KUKA KRL program: MyProgram_305().src

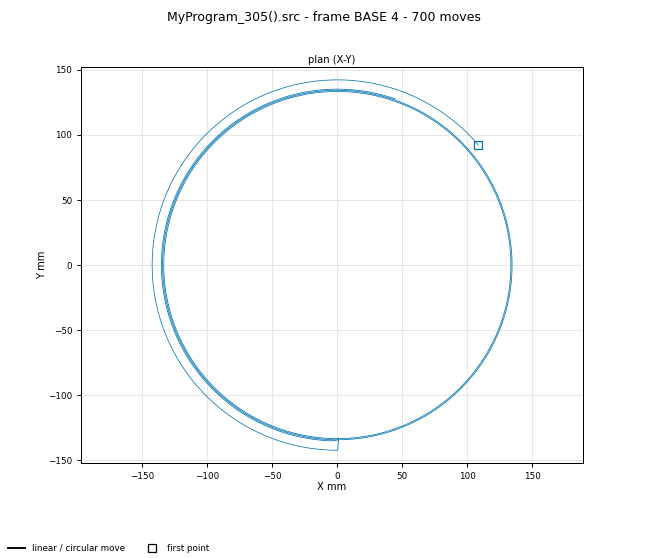
[picture p0: tool path of MyProgram_305().src in frame BASE 4, 700 of 700 moves have a stored position in this frame; points joined in program order, loops and branches not executed]
&ACCESS RVP
&REL 1
&PARAM TEMPLATE = C:\KRC\Roboter\Template\vorgabe
&PARAM EDITMASK = *
DEF MyProgram_305()
; ---- Setting reference (Base) ----
$BASE = BASE_DATA[4]

; --------------------------
; ---- Setting tool (TCP) ----
$TOOL = TOOL_DATA[3]
; --------------------------

$VEL.CP = VEL_APROX_PRINT
Startdeposition()
$VEL.CP = VEL_PRINT
LIN {X 108.497,Y 92.2361,Z 180,A 42.4872,B 5.0785,C 0.1519,E1 5.2028,E2 410.3593} C_DIS
LIN {X 105.629,Y 95.5075,Z 180,A 44.1909,B 5.0786,C 0.1489,E1 5.1996,E2 408.6614} C_DIS
LIN {X 103.133,Y 98.1976,Z 180,A 45.6374,B 5.0786,C 0.1462,E1 5.1969,E2 407.2184} C_DIS
LIN {X 100.1614,Y 101.227,Z 180,A 47.3328,B 5.0788,C 0.1429,E1 5.1935,E2 405.5242} C_DIS
LIN {X 97.4009,Y 103.8864,Z 180,A 48.922,B 5.0788,C 0.1392,E1 5.1903,E2 403.9286} C_DIS
LIN {X 93.8802,Y 107.0781,Z 180,A 50.7517,B 5.079,C 0.1367,E1 5.1865,E2 402.1093} C_DIS
LIN {X 90.8749,Y 109.6397,Z 180,A 52.3365,B 5.079,C 0.1338,E1 5.1831,E2 400.5248} C_DIS
LIN {X 87.4731,Y 112.3728,Z 180,A 54.072,B 5.0791,C 0.1309,E1 5.1793,E2 398.7918} C_DIS
LIN {X 84.1137,Y 114.9089,Z 180,A 55.7406,B 5.0791,C 0.1284,E1 5.1756,E2 397.1263} C_DIS
LIN {X 80.5548,Y 117.431,Z 180,A 57.3714,B 5.0791,C 0.1271,E1 5.1719,E2 395.5116} C_DIS
LIN {X 76.9953,Y 119.7953,Z 180,A 59.0501,B 5.0793,C 0.1249,E1 5.1679,E2 393.8381} C_DIS
LIN {X 73.811,Y 121.7829,Z 180,A 60.6088,B 5.0793,C 0.122,E1 5.1642,E2 392.273} C_DIS
LIN {X 70.1888,Y 123.9065,Z 180,A 62.306,B 5.0793,C 0.1195,E1 5.1601,E2 390.5749} C_DIS
LIN {X 66.4714,Y 125.9372,Z 180,A 63.6729,B 5.0793,C 0.1215,E1 5.1569,E2 389.2516} C_DIS
LIN {X 63.8622,Y 127.2826,Z 180,A 65.0425,B 5.0794,C 0.1175,E1 5.1534,E2 387.8578} C_DIS
LIN {X 60.0878,Y 129.1051,Z 180,A 66.7376,B 5.0794,C 0.1152,E1 5.1491,E2 386.1617} C_DIS
LIN {X 56.1086,Y 130.8838,Z 180,A 68.5245,B 5.0795,C 0.1128,E1 5.1445,E2 384.3707} C_DIS
LIN {X 51.5758,Y 132.7347,Z 180,A 70.4336,B 5.0795,C 0.1114,E1 5.1396,E2 382.4697} C_DIS
LIN {X 47.7101,Y 134.1742,Z 180,A 72.0661,B 5.0795,C 0.11,E1 5.1353,E2 380.841} C_DIS
LIN {X 44.2479,Y 135.3562,Z 180,A 73.5098,B 5.0796,C 0.109,E1 5.1315,E2 379.4014} C_DIS
LIN {X 40.4549,Y 136.5365,Z 180,A 75.105,B 5.0796,C 0.1077,E1 5.1272,E2 377.8068} C_DIS
LIN {X 36.267,Y 137.708,Z 180,A 76.8248,B 5.0796,C 0.1066,E1 5.1226,E2 376.0913} C_DIS
LIN {X 32.5455,Y 138.6366,Z 180,A 78.3403,B 5.0796,C 0.1059,E1 5.1185,E2 374.5798} C_DIS
LIN {X 29.1374,Y 139.3923,Z 180,A 79.7398,B 5.0797,C 0.105,E1 5.1147,E2 373.1814} C_DIS
LIN {X 26.0616,Y 139.9996,Z 180,A 80.976,B 5.0797,C 0.1046,E1 5.1113,E2 371.9487} C_DIS
LIN {X 22.184,Y 140.6651,Z 180,A 82.5487,B 5.0797,C 0.1039,E1 5.107,E2 370.3778} C_DIS
LIN {X 18.7998,Y 141.157,Z 180,A 83.9352,B 5.0797,C 0.1032,E1 5.1031,E2 368.9904} C_DIS
LIN {X 15.3344,Y 141.5752,Z 180,A 85.3305,B 5.0797,C 0.1028,E1 5.0993,E2 367.5967} C_DIS
LIN {X 11.8606,Y 141.9085,Z 180,A 86.7247,B 5.0797,C 0.1025,E1 5.0954,E2 366.2043} C_DIS
LIN {X 8.3796,Y 142.157,Z 180,A 88.0849,B 5.0797,C 0.1027,E1 5.0916,E2 364.8504} C_DIS
LIN {X 5.2259,Y 142.3077,Z 180,A 89.42,B 5.0797,C 0.1017,E1 5.0879,E2 363.5075} C_DIS
LIN {X 0.9091,Y 142.4005,Z 180,A 91.0268,B 5.0797,C 0.103,E1 5.0834,E2 361.9182} C_DIS
LIN {X -1.7521,Y 142.3939,Z 180,A 92.2232,B 5.0797,C 0.1016,E1 5.08,E2 360.7062} C_DIS
LIN {X -5.5962,Y 142.2933,Z 180,A 93.6931,B 5.0797,C 0.1025,E1 5.076,E2 359.2469} C_DIS
LIN {X -8.754,Y 142.1339,Z 180,A 95.0256,B 5.0797,C 0.102,E1 5.0722,E2 357.9071} C_DIS
LIN {X -12.2328,Y 141.877,Z 180,A 96.4261,B 5.0797,C 0.1023,E1 5.0683,E2 356.5077} C_DIS
LIN {X -15.7034,Y 141.5355,Z 180,A 97.8292,B 5.0797,C 0.1026,E1 5.0644,E2 355.1055} C_DIS
LIN {X -19.165,Y 141.1092,Z 180,A 99.3368,B 5.0797,C 0.1019,E1 5.0602,E2 353.5852} C_DIS
LIN {X -23.0175,Y 140.5312,Z 180,A 100.8267,B 5.0797,C 0.1034,E1 5.0561,E2 352.1061} C_DIS
LIN {X -26.1042,Y 139.9915,Z 180,A 102.0941,B 5.0797,C 0.1039,E1 5.0527,E2 350.8385} C_DIS
LIN {X -29.5153,Y 139.3118,Z 180,A 103.4975,B 5.0797,C 0.1046,E1 5.0488,E2 349.4354} C_DIS
LIN {X -33.0361,Y 138.5184,Z 180,A 104.9194,B 5.0797,C 0.1058,E1 5.045,E2 348.0183} C_DIS
LIN {X -36.6145,Y 137.6154,Z 180,A 106.458,B 5.0797,C 0.1062,E1 5.0408,E2 346.4736} C_DIS
LIN {X -40.0082,Y 136.6672,Z 180,A 107.8792,B 5.0797,C 0.1072,E1 5.037,E2 345.0529} C_DIS
LIN {X -43.347,Y 135.6452,Z 180,A 109.2169,B 5.0797,C 0.109,E1 5.0334,E2 343.7247} C_DIS
LIN {X -46.3341,Y 134.6545,Z 180,A 110.6489,B 5.0797,C 0.1084,E1 5.0296,E2 342.2722} C_DIS
LIN {X -49.9691,Y 133.3479,Z 180,A 112.1416,B 5.0796,C 0.1105,E1 5.0257,E2 340.7885} C_DIS
LIN {X -52.8929,Y 132.2159,Z 180,A 113.4133,B 5.0796,C 0.1117,E1 5.0224,E2 339.5163} C_DIS
LIN {X -56.1132,Y 130.8818,Z 180,A 114.9688,B 5.0796,C 0.1116,E1 5.0183,E2 337.942} C_DIS
LIN {X -60.2519,Y 129.0292,Z 180,A 116.7977,B 5.0796,C 0.1136,E1 5.0137,E2 336.1139} C_DIS
LIN {X -64.2345,Y 127.093,Z 180,A 118.4648,B 5.0794,C 0.117,E1 5.0096,E2 334.4628} C_DIS
LIN {X -67.29,Y 125.5037,Z 180,A 119.9727,B 5.0794,C 0.1176,E1 5.0058,E2 332.9403} C_DIS
LIN {X -70.8659,Y 123.5203,Z 180,A 121.6,B 5.0794,C 0.12,E1 5.0019,E2 331.3165} C_DIS
LIN {X -74.4835,Y 121.3727,Z 180,A 123.3149,B 5.0794,C 0.1222,E1 4.9978,E2 329.6} C_DIS
LIN {X -77.8009,Y 119.2738,Z 180,A 124.9752,B 5.0793,C 0.1238,E1 4.9938,E2 327.9305} C_DIS
LIN {X -81.4658,Y 116.8009,Z 180,A 126.8101,B 5.0793,C 0.1261,E1 4.9896,E2 326.0897} C_DIS
LIN {X -85.414,Y 113.9463,Z 180,A 128.7148,B 5.0791,C 0.1298,E1 4.9853,E2 324.1938} C_DIS
LIN {X -88.4535,Y 111.6027,Z 180,A 130.3727,B 5.0791,C 0.1314,E1 4.9817,E2 322.5224} C_DIS
LIN {X -92.2127,Y 108.5169,Z 180,A 132.2804,B 5.079,C 0.1354,E1 4.9776,E2 320.6226} C_DIS
LIN {X -95.5234,Y 105.6146,Z 180,A 134.0811,B 5.079,C 0.1385,E1 4.9738,E2 318.8196} C_DIS
LIN {X -98.7082,Y 102.645,Z 180,A 135.9095,B 5.0788,C 0.1411,E1 4.9701,E2 316.9829} C_DIS
LIN {X -101.7995,Y 99.5791,Z 180,A 137.6842,B 5.0788,C 0.1444,E1 4.9666,E2 315.2066} C_DIS
LIN {X -104.4911,Y 96.7516,Z 180,A 139.363,B 5.0787,C 0.1467,E1 4.9634,E2 313.515} C_DIS
LIN {X -107.2862,Y 93.6417,Z 180,A 140.9733,B 5.0785,C 0.1509,E1 4.9604,E2 311.9156} C_DIS
LIN {X -110.089,Y 90.3304,Z 180,A 142.8502,B 5.0785,C 0.1535,E1 4.957,E2 310.0231} C_DIS
LIN {X -112.7881,Y 86.9374,Z 180,A 144.5372,B 5.0783,C 0.1579,E1 4.9541,E2 308.345} C_DIS
LIN {X -115.4142,Y 83.4188,Z 180,A 146.4481,B 5.0783,C 0.1606,E1 4.9509,E2 306.4169} C_DIS
LIN {X -118.0164,Y 79.6949,Z 180,A 148.3219,B 5.0781,C 0.1645,E1 4.948,E2 304.5386} C_DIS
LIN {X -120.4113,Y 76.0279,Z 180,A 150.0764,B 5.078,C 0.1688,E1 4.9453,E2 302.7867} C_DIS
LIN {X -122.5944,Y 72.456,Z 180,A 151.8564,B 5.0779,C 0.172,E1 4.9428,E2 300.9958} C_DIS
LIN {X -124.8426,Y 68.5097,Z 180,A 153.5741,B 5.0777,C 0.1775,E1 4.9404,E2 299.2939} C_DIS
LIN {X -126.5036,Y 65.3923,Z 180,A 155.0584,B 5.0776,C 0.1805,E1 4.9385,E2 297.8026} C_DIS
LIN {X -128.0663,Y 62.2752,Z 180,A 156.662,B 5.0776,C 0.1824,E1 4.9365,E2 296.174} C_DIS
LIN {X -129.8361,Y 58.4918,Z 180,A 158.3236,B 5.0774,C 0.1869,E1 4.9346,E2 294.5162} C_DIS
LIN {X -131.6971,Y 54.1756,Z 180,A 160.1551,B 5.0772,C 0.1923,E1 4.9326,E2 292.6943} C_DIS
LIN {X -132.8628,Y 51.2461,Z 180,A 161.4663,B 5.077,C 0.1953,E1 4.9313,E2 291.3785} C_DIS
LIN {X -134.0776,Y 47.978,Z 180,A 162.9414,B 5.077,C 0.1985,E1 4.9298,E2 289.8952} C_DIS
LIN {X -135.2171,Y 44.6658,Z 180,A 164.3548,B 5.0768,C 0.2022,E1 4.9286,E2 288.4824} C_DIS
LIN {X -136.271,Y 41.3393,Z 180,A 165.7974,B 5.0766,C 0.2057,E1 4.9274,E2 287.0359} C_DIS
LIN {X -137.2431,Y 37.9877,Z 180,A 167.24,B 5.0765,C 0.2092,E1 4.9263,E2 285.5894} C_DIS
LIN {X -138.2216,Y 34.2642,Z 180,A 168.83,B 5.0763,C 0.2132,E1 4.9252,E2 283.9955} C_DIS
LIN {X -139.0703,Y 30.6335,Z 180,A 170.3234,B 5.0761,C 0.2174,E1 4.9243,E2 282.5042} C_DIS
LIN {X -139.7442,Y 27.3977,Z 180,A 171.7791,B 5.0761,C 0.22,E1 4.9235,E2 281.033} C_DIS
LIN {X -140.3142,Y 24.3143,Z 180,A 173.0378,B 5.0759,C 0.2236,E1 4.9228,E2 279.7758} C_DIS
LIN {X -140.9162,Y 20.5282,Z 180,A 174.6365,B 5.0757,C 0.2274,E1 4.9222,E2 278.1708} C_DIS
LIN {X -141.3751,Y 17.0814,Z 180,A 176.0816,B 5.0755,C 0.231,E1 4.9217,E2 276.7207} C_DIS
LIN {X -141.7543,Y 13.5793,Z 180,A 177.5278,B 5.0754,C 0.2348,E1 4.9212,E2 275.2719} C_DIS
LIN {X -142.0445,Y 10.1047,Z 180,A 178.9648,B 5.0752,C 0.2385,E1 4.9209,E2 273.8315} C_DIS
LIN {X -142.2324,Y 6.9769,Z 180,A -179.6803,B 5.0751,C 0.2412,E1 4.9207,E2 272.4651} C_DIS
LIN {X -142.3708,Y 3.1405,Z 180,A -178.0382,B 5.0749,C 0.2448,E1 4.9207,E2 270.8114} C_DIS
LIN {X -142.4071,Y -0.0245,Z 180,A -176.7476,B 5.0747,C 0.2483,E1 4.9207,E2 269.5195} C_DIS
LIN {X -142.3604,Y -3.5237,Z 180,A -175.2972,B 5.0746,C 0.2519,E1 4.9207,E2 268.0644} C_DIS
LIN {X -142.231,Y -7.0045,Z 180,A -173.9334,B 5.0743,C 0.2562,E1 4.9208,E2 266.7066} C_DIS
LIN {X -142.0173,Y -10.477,Z 180,A -172.4754,B 5.0742,C 0.2597,E1 4.9211,E2 265.2419} C_DIS
LIN {X -141.7082,Y -14.0595,Z 180,A -171.0171,B 5.074,C 0.2637,E1 4.9215,E2 263.7831} C_DIS
LIN {X -141.3237,Y -17.5129,Z 180,A -169.5808,B 5.0738,C 0.2673,E1 4.922,E2 262.3427} C_DIS
LIN {X -140.8041,Y -21.2862,Z 180,A -167.9868,B 5.0736,C 0.271,E1 4.9226,E2 260.7416} C_DIS
LIN {X -140.2364,Y -24.7488,Z 180,A -166.6703,B 5.0733,C 0.2758,E1 4.9232,E2 259.4386} C_DIS
LIN {X -139.6676,Y -27.7843,Z 180,A -165.2521,B 5.0733,C 0.2777,E1 4.924,E2 257.998} C_DIS
LIN {X -138.9437,Y -31.2015,Z 180,A -163.8091,B 5.073,C 0.2813,E1 4.9248,E2 256.5508} C_DIS
LIN {X -138.1369,Y -34.5977,Z 180,A -162.2841,B 5.0729,C 0.2841,E1 4.9259,E2 255.0107} C_DIS
LIN {X -137.1471,Y -38.3311,Z 180,A -160.7717,B 5.0726,C 0.2887,E1 4.927,E2 253.5046} C_DIS
LIN {X -136.1664,Y -41.681,Z 180,A -159.328,B 5.0724,C 0.2921,E1 4.9281,E2 252.0566} C_DIS
LIN {X -135.2162,Y -44.6685,Z 180,A -158.0324,B 5.0722,C 0.2952,E1 4.9293,E2 250.7571} C_DIS
LIN {X -133.9438,Y -48.3491,Z 180,A -156.423,B 5.072,C 0.299,E1 4.9308,E2 249.1429} C_DIS
LIN {X -132.7219,Y -51.6087,Z 180,A -155.0665,B 5.0718,C 0.3031,E1 4.9321,E2 247.793} C_DIS
LIN {X -131.5581,Y -54.5086,Z 180,A -153.6984,B 5.0716,C 0.3054,E1 4.9336,E2 246.4108} C_DIS
LIN {X -130.1902,Y -57.7,Z 180,A -152.2583,B 5.0714,C 0.3086,E1 4.9352,E2 244.9656} C_DIS
LIN {X -128.7297,Y -60.8892,Z 180,A -150.8166,B 5.0712,C 0.3119,E1 4.9369,E2 243.5205} C_DIS
LIN {X -127.1988,Y -64.0267,Z 180,A -149.3238,B 5.0711,C 0.3146,E1 4.9387,E2 242.0166} C_DIS
LIN {X -125.4914,Y -67.313,Z 180,A -147.7585,B 5.0709,C 0.3176,E1 4.9408,E2 240.4419} C_DIS
LIN {X -123.3746,Y -71.1188,Z 180,A -145.9254,B 5.0707,C 0.3211,E1 4.9433,E2 238.5986} C_DIS
LIN {X -121.1439,Y -74.8563,Z 180,A -144.1142,B 5.0704,C 0.3247,E1 4.946,E2 236.7801} C_DIS
LIN {X -118.8861,Y -78.3915,Z 180,A -142.4947,B 5.0701,C 0.3293,E1 4.9484,E2 235.1704} C_DIS
LIN {X -116.4277,Y -81.9983,Z 180,A -140.6547,B 5.0699,C 0.3325,E1 4.9514,E2 233.3197} C_DIS
LIN {X -113.8558,Y -85.534,Z 180,A -138.8009,B 5.0697,C 0.3356,E1 4.9545,E2 231.4538} C_DIS
LIN {X -111.0721,Y -89.1192,Z 180,A -136.9271,B 5.0695,C 0.3391,E1 4.9577,E2 229.5741} C_DIS
LIN {X -108.1727,Y -92.6172,Z 180,A -135.0822,B 5.0692,C 0.3428,E1 4.9611,E2 227.7274} C_DIS
LIN {X -105.043,Y -96.1518,Z 180,A -133.218,B 5.069,C 0.347,E1 4.9645,E2 225.8684} C_DIS
LIN {X -102.3499,Y -99.0132,Z 180,A -131.546,B 5.0688,C 0.3492,E1 4.9678,E2 224.1844} C_DIS
LIN {X -98.9579,Y -102.4034,Z 180,A -129.6209,B 5.0685,C 0.353,E1 4.9716,E2 222.2603} C_DIS
LIN {X -95.6326,Y -105.5155,Z 180,A -127.7753,B 5.0683,C 0.3562,E1 4.9754,E2 220.4133} C_DIS
LIN {X -92.4851,Y -108.2854,Z 180,A -126.016,B 5.0682,C 0.3585,E1 4.9791,E2 218.6444} C_DIS
LIN {X -88.9817,Y -111.1824,Z 180,A -124.179,B 5.0679,C 0.3616,E1 4.9831,E2 216.8065} C_DIS
LIN {X -85.5169,Y -113.8687,Z 180,A -122.4297,B 5.0677,C 0.3646,E1 4.987,E2 215.0594} C_DIS
LIN {X -82.7018,Y -115.929,Z 180,A -120.8841,B 5.0677,C 0.3653,E1 4.9906,E2 213.4946} C_DIS
LIN {X -78.9676,Y -118.5042,Z 180,A -119.1549,B 5.0674,C 0.3691,E1 4.9945,E2 211.7785} C_DIS
LIN {X -75.4545,Y -120.7717,Z 180,A -117.4099,B 5.0673,C 0.3708,E1 4.9987,E2 210.025} C_DIS
LIN {X -71.7041,Y -123.0358,Z 180,A -115.6316,B 5.0671,C 0.373,E1 5.0029,E2 208.2445} C_DIS
LIN {X -68.4223,Y -124.8903,Z 180,A -114.1736,B 5.0669,C 0.3756,E1 5.0065,E2 206.7944} C_DIS
LIN {X -65.4161,Y -126.4913,Z 180,A -112.7306,B 5.0669,C 0.3765,E1 5.0101,E2 205.3415} C_DIS
LIN {X -62.2971,Y -128.0555,Z 180,A -111.1595,B 5.0669,C 0.3763,E1 5.0141,E2 203.7473} C_DIS
LIN {X -58.3478,Y -129.9004,Z 180,A -109.479,B 5.0667,C 0.379,E1 5.0183,E2 202.0767} C_DIS
LIN {X -54.1627,Y -131.7025,Z 180,A -107.7004,B 5.0665,C 0.3814,E1 5.0229,E2 200.3054} C_DIS
LIN {X -51.0763,Y -132.9289,Z 180,A -106.3426,B 5.0665,C 0.3824,E1 5.0264,E2 198.9443} C_DIS
LIN {X -47.7687,Y -134.1531,Z 180,A -104.8979,B 5.0663,C 0.3833,E1 5.0302,E2 197.4959} C_DIS
LIN {X -44.4743,Y -135.2809,Z 180,A -103.5072,B 5.0663,C 0.3845,E1 5.0339,E2 196.1064} C_DIS
LIN {X -41.0445,Y -136.3612,Z 180,A -102.061,B 5.0662,C 0.3856,E1 5.0378,E2 194.6599} C_DIS
LIN {X -37.9589,Y -137.2512,Z 180,A -100.7471,B 5.0662,C 0.3861,E1 5.0413,E2 193.3426} C_DIS
LIN {X -34.247,Y -138.2259,Z 180,A -99.1966,B 5.0661,C 0.387,E1 5.0455,E2 191.7909} C_DIS
LIN {X -30.8491,Y -139.0238,Z 180,A -97.7718,B 5.0661,C 0.3874,E1 5.0494,E2 190.3629} C_DIS
LIN {X -27.4327,Y -139.7375,Z 180,A -96.4289,B 5.0659,C 0.3888,E1 5.053,E2 189.0279} C_DIS
LIN {X -24.3325,Y -140.3109,Z 180,A -95.1056,B 5.0659,C 0.3886,E1 5.0567,E2 187.6967} C_DIS
LIN {X -20.5341,Y -140.9154,Z 180,A -93.538,B 5.0659,C 0.3888,E1 5.061,E2 186.1258} C_DIS
LIN {X -17.0731,Y -141.3761,Z 180,A -92.1332,B 5.0659,C 0.3892,E1 5.0649,E2 184.7205} C_DIS
LIN {X -13.6034,Y -141.752,Z 180,A -90.7314,B 5.0659,C 0.3894,E1 5.0688,E2 183.3185} C_DIS
LIN {X -10.1088,Y -142.0442,Z 180,A -89.3263,B 5.0659,C 0.3896,E1 5.0727,E2 181.9136} C_DIS
LIN {X -6.975,Y -142.2325,Z 180,A -88.0242,B 5.0659,C 0.3892,E1 5.0764,E2 180.6056} C_DIS
LIN {X -3.1346,Y -142.3709,Z 180,A -86.5457,B 5.0659,C 0.3899,E1 5.0805,E2 179.1357} C_DIS
LIN {X 0.3576,Y -142.4035,Z 180,A -85.1921,B 5.0659,C 0.3904,E1 5.0843,E2 177.7885} C_DIS
LIN {X 0.3576,Y -142.4035,Z 180,A -85.1921,B 5.0659,C 0.3904,E1 5.0843,E2 177.7885} C_DIS
Enddeposition()
LIN {X 0.9666,Y -133.4651,Z 181,A -85.2276,B 5.1404,C 0.3663,E1 5.1577,E2 177.5189} C_DIS
Startdeposition()
$VEL.CP = VEL_PRINT
LIN {X -2.5839,Y -133.4454,Z 181,A -87.4468,B 5.1398,C 0.3744,E1 5.1512,E2 179.8265} C_DIS
LIN {X -7.4832,Y -133.2619,Z 181,A -89.3757,B 5.14,C 0.3724,E1 5.1459,E2 181.7343} C_DIS
LIN {X -10.7403,Y -133.0379,Z 181,A -90.8246,B 5.14,C 0.3728,E1 5.1419,E2 183.1897} C_DIS
LIN {X -13.9556,Y -132.7386,Z 181,A -92.3357,B 5.1399,C 0.374,E1 5.1376,E2 184.717} C_DIS
LIN {X -17.9739,Y -132.2555,Z 181,A -93.9306,B 5.14,C 0.372,E1 5.1332,E2 186.2947} C_DIS
LIN {X -21.21,Y -131.7759,Z 181,A -95.3324,B 5.14,C 0.3716,E1 5.1294,E2 187.6966} C_DIS
LIN {X -25.2351,Y -131.0625,Z 181,A -97.1246,B 5.14,C 0.3713,E1 5.1244,E2 189.4941} C_DIS
LIN {X -29.2391,Y -130.2285,Z 181,A -98.8863,B 5.1401,C 0.3705,E1 5.1196,E2 191.257} C_DIS
LIN {X -33.132,Y -129.2923,Z 181,A -100.6252,B 5.1401,C 0.3698,E1 5.1149,E2 192.999} C_DIS
LIN {X -36.6436,Y -128.3429,Z 181,A -102.1754,B 5.1403,C 0.3687,E1 5.1107,E2 194.5482} C_DIS
LIN {X -39.6132,Y -127.4568,Z 181,A -103.5231,B 5.1403,C 0.3679,E1 5.1071,E2 195.8983} C_DIS
LIN {X -42.7923,Y -126.4253,Z 181,A -104.963,B 5.1403,C 0.3668,E1 5.1033,E2 197.3391} C_DIS
LIN {X -45.8064,Y -125.3643,Z 181,A -106.3383,B 5.1405,C 0.3657,E1 5.0997,E2 198.7152} C_DIS
LIN {X -48.9062,Y -124.1879,Z 181,A -107.7863,B 5.1405,C 0.3647,E1 5.0959,E2 200.1665} C_DIS
LIN {X -51.9332,Y -122.9525,Z 181,A -109.3465,B 5.1405,C 0.3649,E1 5.0918,E2 201.7464} C_DIS
LIN {X -55.582,Y -121.3464,Z 181,A -110.979,B 5.1407,C 0.3623,E1 5.0877,E2 203.3693} C_DIS
LIN {X -59.1813,Y -119.6314,Z 181,A -112.6628,B 5.1409,C 0.3601,E1 5.0835,E2 205.0497} C_DIS
LIN {X -62.0962,Y -118.1445,Z 181,A -114.0309,B 5.141,C 0.358,E1 5.0801,E2 206.4134} C_DIS
LIN {X -65.1789,Y -116.4748,Z 181,A -115.6023,B 5.141,C 0.3568,E1 5.0762,E2 207.9933} C_DIS
LIN {X -68.6256,Y -114.4782,Z 181,A -117.3443,B 5.1412,C 0.3548,E1 5.072,E2 209.7393} C_DIS
LIN {X -71.4102,Y -112.7619,Z 181,A -118.7665,B 5.1413,C 0.353,E1 5.0686,E2 211.1637} C_DIS
LIN {X -74.1524,Y -110.9776,Z 181,A -120.1893,B 5.1415,C 0.3511,E1 5.0653,E2 212.5887} C_DIS
LIN {X -76.849,Y -109.1277,Z 181,A -121.6122,B 5.1416,C 0.3492,E1 5.062,E2 214.014} C_DIS
LIN {X -80.0734,Y -106.785,Z 181,A -123.463,B 5.1417,C 0.3477,E1 5.0578,E2 215.8821} C_DIS
LIN {X -83.4049,Y -104.2035,Z 181,A -125.2703,B 5.1419,C 0.3447,E1 5.0539,E2 217.6889} C_DIS
LIN {X -86.7642,Y -101.4237,Z 181,A -127.2201,B 5.1421,C 0.3421,E1 5.0497,E2 219.6481} C_DIS
LIN {X -89.9135,Y -98.6421,Z 181,A -129.0282,B 5.1423,C 0.3389,E1 5.0459,E2 221.4565} C_DIS
LIN {X -92.8898,Y -95.8442,Z 181,A -130.7944,B 5.1425,C 0.3357,E1 5.0423,E2 223.2239} C_DIS
LIN {X -96.0008,Y -92.728,Z 181,A -132.7649,B 5.1427,C 0.3327,E1 5.0385,E2 225.204} C_DIS
LIN {X -98.8906,Y -89.6397,Z 181,A -134.5787,B 5.1429,C 0.329,E1 5.035,E2 227.0171} C_DIS
LIN {X -101.5992,Y -86.5577,Z 181,A -136.389,B 5.1431,C 0.3258,E1 5.0317,E2 228.833} C_DIS
LIN {X -104.1703,Y -83.4465,Z 181,A -138.1887,B 5.1433,C 0.3227,E1 5.0285,E2 230.6405} C_DIS
LIN {X -106.7734,Y -80.0887,Z 181,A -139.9426,B 5.1436,C 0.3181,E1 5.0256,E2 232.3851} C_DIS
LIN {X -109.129,Y -76.8471,Z 181,A -141.5517,B 5.1439,C 0.3132,E1 5.023,E2 233.9799} C_DIS
LIN {X -110.581,Y -74.7426,Z 181,A -142.819,B 5.1439,C 0.3122,E1 5.0209,E2 235.2678} C_DIS
LIN {X -112.3784,Y -72.0119,Z 181,A -144.2543,B 5.1442,C 0.3091,E1 5.0187,E2 236.7065} C_DIS
LIN {X -114.1093,Y -69.2367,Z 181,A -145.7239,B 5.1443,C 0.3064,E1 5.0166,E2 238.1836} C_DIS
LIN {X -116.1638,Y -65.7323,Z 181,A -147.4769,B 5.1446,C 0.3022,E1 5.0141,E2 239.937} C_DIS
LIN {X -117.724,Y -62.8949,Z 181,A -148.9275,B 5.1447,C 0.2993,E1 5.0122,E2 241.3944} C_DIS
LIN {X -119.2188,Y -60.0109,Z 181,A -150.327,B 5.1449,C 0.2959,E1 5.0104,E2 242.794} C_DIS
LIN {X -120.6574,Y -57.0626,Z 181,A -151.7847,B 5.1451,C 0.2927,E1 5.0086,E2 244.257} C_DIS
LIN {X -122.0201,Y -54.0867,Z 181,A -153.225,B 5.1453,C 0.2894,E1 5.007,E2 245.7009} C_DIS
LIN {X -123.3091,Y -51.0793,Z 181,A -154.6658,B 5.1455,C 0.2861,E1 5.0054,E2 247.1454} C_DIS
LIN {X -124.5313,Y -48.0227,Z 181,A -156.1156,B 5.1457,C 0.2827,E1 5.0039,E2 248.5989} C_DIS
LIN {X -125.9117,Y -44.2797,Z 181,A -157.8719,B 5.1459,C 0.2785,E1 5.0023,E2 250.3596} C_DIS
LIN {X -126.9576,Y -41.1855,Z 181,A -159.3753,B 5.1461,C 0.2755,E1 5.0009,E2 251.8746} C_DIS
LIN {X -128.1864,Y -37.1818,Z 181,A -161.2845,B 5.1463,C 0.2715,E1 4.9994,E2 253.7963} C_DIS
LIN {X -129.2875,Y -33.151,Z 181,A -163.0071,B 5.1466,C 0.2661,E1 4.9982,E2 255.5091} C_DIS
LIN {X -130.1807,Y -29.4485,Z 181,A -164.7066,B 5.1468,C 0.2621,E1 4.9971,E2 257.2155} C_DIS
LIN {X -130.9066,Y -26.0376,Z 181,A -166.2181,B 5.147,C 0.2581,E1 4.9962,E2 258.7278} C_DIS
LIN {X -131.5065,Y -22.8186,Z 181,A -167.6603,B 5.1472,C 0.2544,E1 4.9955,E2 260.1737} C_DIS
LIN {X -132.1563,Y -18.6798,Z 181,A -169.4876,B 5.1474,C 0.2496,E1 4.9947,E2 262.0032} C_DIS
LIN {X -132.5766,Y -15.4201,Z 181,A -171.1167,B 5.1474,C 0.2473,E1 4.9942,E2 263.6578} C_DIS
LIN {X -133.0382,Y -10.7366,Z 181,A -173.0667,B 5.1478,C 0.2411,E1 4.9937,E2 265.5978} C_DIS
LIN {X -133.2626,Y -7.4715,Z 181,A -174.576,B 5.1479,C 0.2379,E1 4.9934,E2 267.1188} C_DIS
LIN {X -133.4086,Y -4.0606,Z 181,A -176.1459,B 5.1481,C 0.2345,E1 4.9933,E2 268.7002} C_DIS
LIN {X -133.471,Y -0.1546,Z 181,A -177.6609,B 5.1484,C 0.2285,E1 4.9933,E2 270.1944} C_DIS
LIN {X -133.4459,Y 2.559,Z 181,A -179.0776,B 5.1484,C 0.2272,E1 4.9933,E2 271.6406} C_DIS
LIN {X -133.2634,Y 7.4588,Z 181,A 178.9282,B 5.1487,C 0.2203,E1 4.9935,E2 273.6199} C_DIS
LIN {X -133.0792,Y 10.2167,Z 181,A 177.5657,B 5.1488,C 0.2183,E1 4.9938,E2 275.0026} C_DIS
LIN {X -132.6571,Y 14.7129,Z 181,A 175.6954,B 5.1491,C 0.2123,E1 4.9943,E2 276.8631} C_DIS
LIN {X -132.2572,Y 17.9613,Z 181,A 174.2524,B 5.1492,C 0.2086,E1 4.9949,E2 278.3096} C_DIS
LIN {X -131.7782,Y 21.1963,Z 181,A 172.8099,B 5.1494,C 0.205,E1 4.9955,E2 279.7557} C_DIS
LIN {X -131.0459,Y 25.3219,Z 181,A 170.9461,B 5.1495,C 0.2004,E1 4.9964,E2 281.6259} C_DIS
LIN {X -130.2225,Y 29.2653,Z 181,A 169.1614,B 5.1497,C 0.196,E1 4.9975,E2 283.4158} C_DIS
LIN {X -129.289,Y 33.1449,Z 181,A 167.3853,B 5.1499,C 0.1918,E1 4.9987,E2 285.198} C_DIS
LIN {X -128.1873,Y 37.1787,Z 181,A 165.4197,B 5.1499,C 0.1882,E1 5.0002,E2 287.1825} C_DIS
LIN {X -126.959,Y 41.1809,Z 181,A 163.7112,B 5.1502,C 0.1826,E1 5.0016,E2 288.8789} C_DIS
LIN {X -125.9133,Y 44.2753,Z 181,A 162.2771,B 5.1503,C 0.1791,E1 5.0029,E2 290.3157} C_DIS
LIN {X -124.8551,Y 47.1748,Z 181,A 160.8879,B 5.1504,C 0.1761,E1 5.0042,E2 291.7113} C_DIS
LIN {X -123.5866,Y 50.4058,Z 181,A 159.3862,B 5.1506,C 0.1722,E1 5.0058,E2 293.2132} C_DIS
LIN {X -122.3894,Y 53.2448,Z 181,A 157.9942,B 5.1506,C 0.1693,E1 5.0073,E2 294.6123} C_DIS
LIN {X -120.6575,Y 57.0624,Z 181,A 156.0942,B 5.1508,C 0.1654,E1 5.0096,E2 296.5227} C_DIS
LIN {X -118.8877,Y 60.6613,Z 181,A 154.4056,B 5.1509,C 0.1608,E1 5.0117,E2 298.2059} C_DIS
LIN {X -117.2734,Y 63.7307,Z 181,A 152.8842,B 5.151,C 0.1573,E1 5.0137,E2 299.73} C_DIS
LIN {X -115.6804,Y 66.5791,Z 181,A 151.3012,B 5.151,C 0.1553,E1 5.0159,E2 301.3335} C_DIS
LIN {X -113.6413,Y 70.0023,Z 181,A 149.6873,B 5.1512,C 0.1504,E1 5.0182,E2 302.9344} C_DIS
LIN {X -111.8949,Y 72.7609,Z 181,A 148.2543,B 5.1513,C 0.1473,E1 5.0204,E2 304.3699} C_DIS
LIN {X -110.0603,Y 75.5072,Z 181,A 146.8037,B 5.1514,C 0.1442,E1 5.0226,E2 305.8232} C_DIS
LIN {X -108.1693,Y 78.1923,Z 181,A 145.3636,B 5.1514,C 0.1412,E1 5.025,E2 307.2657} C_DIS
LIN {X -106.221,Y 80.8197,Z 181,A 143.8414,B 5.1516,C 0.139,E1 5.0276,E2 308.8006} C_DIS
LIN {X -103.6931,Y 84.0383,Z 181,A 142.0294,B 5.1516,C 0.1356,E1 5.0307,E2 310.6176} C_DIS
LIN {X -101.06,Y 87.1866,Z 181,A 140.268,B 5.1517,C 0.1318,E1 5.0339,E2 312.3775} C_DIS
LIN {X -98.341,Y 90.2422,Z 181,A 138.4627,B 5.1518,C 0.1285,E1 5.0373,E2 314.1872} C_DIS
LIN {X -95.5305,Y 93.2129,Z 181,A 136.6586,B 5.1519,C 0.1253,E1 5.0408,E2 315.9956} C_DIS
LIN {X -92.6287,Y 96.0969,Z 181,A 134.8509,B 5.1519,C 0.1223,E1 5.0444,E2 317.8079} C_DIS
LIN {X -89.6302,Y 98.8991,Z 181,A 133.0781,B 5.1521,C 0.119,E1 5.048,E2 319.5805} C_DIS
LIN {X -86.5579,Y 101.599,Z 181,A 131.2764,B 5.1521,C 0.1162,E1 5.0519,E2 321.3862} C_DIS
LIN {X -83.4037,Y 104.2044,Z 181,A 129.4735,B 5.1521,C 0.1135,E1 5.0558,E2 323.1932} C_DIS
LIN {X -80.2142,Y 106.6787,Z 181,A 127.7852,B 5.1522,C 0.1101,E1 5.0595,E2 324.8748} C_DIS
LIN {X -77.4818,Y 108.6794,Z 181,A 126.308,B 5.1522,C 0.108,E1 5.0629,E2 326.3537} C_DIS
LIN {X -74.6795,Y 110.6238,Z 181,A 124.8485,B 5.1523,C 0.1056,E1 5.0662,E2 327.8115} C_DIS
LIN {X -71.9747,Y 112.4022,Z 181,A 123.4398,B 5.1523,C 0.1037,E1 5.0695,E2 329.2214} C_DIS
LIN {X -69.2174,Y 114.121,Z 181,A 122.0267,B 5.1524,C 0.1018,E1 5.0729,E2 330.6356} C_DIS
LIN {X -65.7952,Y 116.1282,Z 181,A 120.3052,B 5.1524,C 0.0996,E1 5.077,E2 332.3581} C_DIS
LIN {X -62.9074,Y 117.7173,Z 181,A 118.8365,B 5.1524,C 0.0982,E1 5.0807,E2 333.832} C_DIS
LIN {X -60.0043,Y 119.2222,Z 181,A 117.4318,B 5.1525,C 0.0965,E1 5.0842,E2 335.2357} C_DIS
LIN {X -56.4138,Y 120.9617,Z 181,A 115.5862,B 5.1525,C 0.0957,E1 5.0889,E2 337.0957} C_DIS
LIN {X -52.5791,Y 122.6772,Z 181,A 113.8788,B 5.1525,C 0.0928,E1 5.0932,E2 338.7906} C_DIS
LIN {X -49.5073,Y 123.9488,Z 181,A 112.439,B 5.1526,C 0.0914,E1 5.0969,E2 340.2309} C_DIS
LIN {X -46.4779,Y 125.1161,Z 181,A 111.0321,B 5.1526,C 0.0902,E1 5.1006,E2 341.6384} C_DIS
LIN {X -42.7332,Y 126.445,Z 181,A 109.3149,B 5.1526,C 0.0888,E1 5.1051,E2 343.3559} C_DIS
LIN {X -39.4514,Y 127.5064,Z 181,A 107.67,B 5.1526,C 0.0891,E1 5.1096,E2 345.019} C_DIS
LIN {X -34.9007,Y 128.8268,Z 181,A 105.711,B 5.1526,C 0.0869,E1 5.1148,E2 346.9681} C_DIS
LIN {X -31.5367,Y 129.6906,Z 181,A 104.2667,B 5.1527,C 0.0855,E1 5.1187,E2 348.406} C_DIS
LIN {X -27.6296,Y 130.5797,Z 181,A 102.545,B 5.1527,C 0.0845,E1 5.1234,E2 350.1268} C_DIS
LIN {X -24.6043,Y 131.1831,Z 181,A 101.2024,B 5.1527,C 0.0841,E1 5.1271,E2 351.4708} C_DIS
LIN {X -21.198,Y 131.7779,Z 181,A 99.7324,B 5.1527,C 0.0833,E1 5.1311,E2 352.9384} C_DIS
LIN {X -17.2518,Y 132.3501,Z 181,A 97.9714,B 5.1527,C 0.0833,E1 5.136,E2 354.7042} C_DIS
LIN {X -13.0669,Y 132.829,Z 181,A 96.0609,B 5.1527,C 0.0838,E1 5.1413,E2 356.6258} C_DIS
LIN {X -8.8889,Y 133.1753,Z 181,A 94.4349,B 5.1527,C 0.0817,E1 5.1458,E2 358.2305} C_DIS
LIN {X -5.8122,Y 133.3447,Z 181,A 92.8722,B 5.1527,C 0.0841,E1 5.1502,E2 359.8208} C_DIS
LIN {X -1.618,Y 133.4615,Z 181,A 91.2767,B 5.1527,C 0.0819,E1 5.1546,E2 361.3913} C_DIS
LIN {X 1.6519,Y 133.4609,Z 181,A 89.8376,B 5.1527,C 0.0824,E1 5.1587,E2 362.834} C_DIS
LIN {X 5.6387,Y 133.3515,Z 181,A 88.142,B 5.1527,C 0.0824,E1 5.1634,E2 364.5269} C_DIS
LIN {X 8.9026,Y 133.1745,Z 181,A 86.681,B 5.1527,C 0.0834,E1 5.1675,E2 365.9942} C_DIS
LIN {X 12.385,Y 132.8945,Z 181,A 85.2419,B 5.1527,C 0.0831,E1 5.1715,E2 367.4256} C_DIS
LIN {X 16.3461,Y 132.4661,Z 181,A 83.557,B 5.1527,C 0.0835,E1 5.1761,E2 369.1069} C_DIS
LIN {X 19.5886,Y 132.0264,Z 181,A 82.1553,B 5.1527,C 0.0841,E1 5.18,E2 370.5078} C_DIS
LIN {X 23.7206,Y 131.3451,Z 181,A 80.3607,B 5.1527,C 0.085,E1 5.1849,E2 372.3014} C_DIS
LIN {X 26.9337,Y 130.7243,Z 181,A 78.8318,B 5.1527,C 0.0872,E1 5.1892,E2 373.8445} C_DIS
LIN {X 30.6668,Y 129.9003,Z 181,A 77.273,B 5.1527,C 0.0874,E1 5.1934,E2 375.3932} C_DIS
LIN {X 33.8696,Y 129.1018,Z 181,A 75.9746,B 5.1527,C 0.0871,E1 5.1969,E2 376.6773} C_DIS
LIN {X 37.2684,Y 128.161,Z 181,A 74.4323,B 5.1527,C 0.0887,E1 5.201,E2 378.2226} C_DIS
LIN {X 40.7299,Y 127.1031,Z 181,A 72.8251,B 5.1527,C 0.0907,E1 5.2053,E2 379.8358} C_DIS
LIN {X 44.3074,Y 125.9021,Z 181,A 71.277,B 5.1527,C 0.0914,E1 5.2094,E2 381.3751} C_DIS
LIN {X 47.1874,Y 124.8503,Z 181,A 69.9555,B 5.1526,C 0.0928,E1 5.2129,E2 382.6971} C_DIS
LIN {X 50.4187,Y 123.5814,Z 181,A 68.4985,B 5.1526,C 0.094,E1 5.2166,E2 384.15} C_DIS
LIN {X 53.2461,Y 122.3888,Z 181,A 67.1738,B 5.1526,C 0.0957,E1 5.22,E2 385.4753} C_DIS
LIN {X 56.4113,Y 120.9629,Z 181,A 65.7442,B 5.1526,C 0.0967,E1 5.2236,E2 386.8977} C_DIS
LIN {X 59.1779,Y 119.6331,Z 181,A 64.4219,B 5.1525,C 0.0985,E1 5.227,E2 388.2203} C_DIS
LIN {X 62.1046,Y 118.1401,Z 181,A 63.0513,B 5.1525,C 0.0999,E1 5.2303,E2 389.5861} C_DIS
LIN {X 65.1756,Y 116.4767,Z 181,A 61.5589,B 5.1525,C 0.1019,E1 5.234,E2 391.0778} C_DIS
LIN {X 68.6226,Y 114.48,Z 181,A 59.8643,B 5.1524,C 0.1042,E1 5.2381,E2 392.7705} C_DIS
LIN {X 71.407,Y 112.7639,Z 181,A 58.4835,B 5.1524,C 0.1061,E1 5.2413,E2 394.1486} C_DIS
LIN {X 74.1476,Y 110.9808,Z 181,A 57.104,B 5.1523,C 0.108,E1 5.2446,E2 395.5253} C_DIS
LIN {X 76.8459,Y 109.1299,Z 181,A 55.5917,B 5.1523,C 0.1117,E1 5.2481,E2 397.0504} C_DIS
LIN {X 80.5688,Y 106.4111,Z 181,A 53.7287,B 5.1522,C 0.1137,E1 5.2522,E2 398.8999} C_DIS
LIN {X 83.6795,Y 103.9826,Z 181,A 52.0272,B 5.1522,C 0.1168,E1 5.2559,E2 400.6024} C_DIS
LIN {X 86.8318,Y 101.3655,Z 181,A 50.2825,B 5.152,C 0.1199,E1 5.2596,E2 402.3456} C_DIS
LIN {X 89.9139,Y 98.6417,Z 181,A 48.5621,B 5.152,C 0.1227,E1 5.2632,E2 404.0609} C_DIS
LIN {X 92.8871,Y 95.8468,Z 181,A 46.8646,B 5.1519,C 0.1254,E1 5.2666,E2 405.7523} C_DIS
LIN {X 95.9897,Y 92.7394,Z 181,A 44.9709,B 5.1519,C 0.1294,E1 5.2703,E2 407.6475} C_DIS
LIN {X 98.8967,Y 89.6328,Z 181,A 43.2263,B 5.1517,C 0.1322,E1 5.2736,E2 409.3828} C_DIS
LIN {X 101.6042,Y 86.5518,Z 181,A 41.491,B 5.1517,C 0.1357,E1 5.2768,E2 411.1155} C_DIS
LIN {X 104.2055,Y 83.4024,Z 181,A 39.7604,B 5.1515,C 0.1392,E1 5.2798,E2 412.8439} C_DIS
LIN {X 106.7752,Y 80.0863,Z 181,A 38.0872,B 5.1515,C 0.1416,E1 5.2827,E2 414.5023} C_DIS
LIN {X 108.5994,Y 77.5937,Z 181,A 36.7653,B 5.1514,C 0.1446,E1 5.2848,E2 415.8242} C_DIS
LIN {X 110.58,Y 74.7441,Z 181,A 35.3438,B 5.1514,C 0.1472,E1 5.287,E2 417.238} C_DIS
LIN {X 112.3765,Y 72.0149,Z 181,A 33.9754,B 5.1512,C 0.1501,E1 5.2891,E2 418.6029} C_DIS
LIN {X 114.1078,Y 69.2391,Z 181,A 32.6065,B 5.1512,C 0.1531,E1 5.2911,E2 419.968} C_DIS
LIN {X 116.1263,Y 65.7985,Z 181,A 30.9487,B 5.1511,C 0.1565,E1 5.2934,E2 421.6201} C_DIS
LIN {X 117.7097,Y 62.9216,Z 181,A 29.5314,B 5.1509,C 0.1602,E1 5.2953,E2 423.0388} C_DIS
LIN {X 119.2226,Y 60.0034,Z 181,A 28.173,B 5.1509,C 0.163,E1 5.297,E2 424.3916} C_DIS
LIN {X 120.657,Y 57.0633,Z 181,A 26.8051,B 5.1508,C 0.1661,E1 5.2987,E2 425.7557} C_DIS
LIN {X 122.0193,Y 54.0884,Z 181,A 25.4371,B 5.1506,C 0.1693,E1 5.3003,E2 427.1199} C_DIS
LIN {X 123.382,Y 50.9048,Z 181,A 23.9932,B 5.1506,C 0.1726,E1 5.3018,E2 428.5595} C_DIS
LIN {X 124.55,Y 47.9746,Z 181,A 22.6728,B 5.1504,C 0.1757,E1 5.3032,E2 429.8765} C_DIS
LIN {X 125.6743,Y 44.9465,Z 181,A 21.3221,B 5.1504,C 0.1789,E1 5.3045,E2 431.2235} C_DIS
LIN {X 126.8507,Y 41.5147,Z 181,A 19.6742,B 5.1501,C 0.1844,E1 5.3059,E2 432.8834} C_DIS
LIN {X 128.1887,Y 37.1739,Z 181,A 17.7855,B 5.15,C 0.1888,E1 5.3074,E2 434.7657} C_DIS
LIN {X 129.2923,Y 33.132,Z 181,A 16.1516,B 5.1499,C 0.1915,E1 5.3086,E2 436.3808} C_DIS
LIN {X 130.2287,Y 29.238,Z 181,A 14.3369,B 5.1496,C 0.1976,E1 5.3097,E2 438.2082} C_DIS
LIN {X 131.0439,Y 25.3324,Z 181,A 12.8113,B 5.1496,C 0.1997,E1 5.3106,E2 439.712} C_DIS
LIN {X 131.6252,Y 22.1134,Z 181,A 11.4412,B 5.1494,C 0.2032,E1 5.3112,E2 441.079} C_DIS
LIN {X 132.1594,Y 18.6582,Z 181,A 10.0202,B 5.1494,C 0.2063,E1 5.3118,E2 442.4912} C_DIS
LIN {X 132.5771,Y 15.416,Z 181,A 8.4862,B 5.1491,C 0.2121,E1 5.3123,E2 444.0421} C_DIS
LIN {X 133.0382,Y 10.7368,Z 181,A 6.6475,B 5.1489,C 0.2153,E1 5.3128,E2 445.8604} C_DIS
LIN {X 133.2391,Y 7.853,Z 181,A 5.3415,B 5.1487,C 0.2197,E1 5.313,E2 447.1751} C_DIS
LIN {X 133.411,Y 3.9751,Z 181,A 3.7211,B 5.1486,C 0.2238,E1 5.3132,E2 448.7911} C_DIS
LIN {X 133.471,Y 0.1531,Z 181,A 2.2813,B 5.1485,C 0.2256,E1 5.3132,E2 450.2076} C_DIS
LIN {X 133.4305,Y -3.2744,Z 181,A 0.6701,B 5.1482,C 0.2318,E1 5.3132,E2 451.837} C_DIS
LIN {X 133.2616,Y -7.4882,Z 181,A -0.9209,B 5.1482,C 0.2339,E1 5.3129,E2 453.4026} C_DIS
LIN {X 133.0374,Y -10.7464,Z 181,A -2.3314,B 5.1479,C 0.238,E1 5.3126,E2 454.8151} C_DIS
LIN {X 132.6571,Y -14.7131,Z 181,A -3.9749,B 5.1478,C 0.2419,E1 5.3122,E2 456.4518} C_DIS
LIN {X 132.2574,Y -17.9595,Z 181,A -5.3383,B 5.1476,C 0.2453,E1 5.3117,E2 457.8113} C_DIS
LIN {X 131.7786,Y -21.1937,Z 181,A -6.7029,B 5.1474,C 0.2487,E1 5.3111,E2 459.1723} C_DIS
LIN {X 131.0432,Y -25.3362,Z 181,A -8.4701,B 5.1472,C 0.2532,E1 5.3102,E2 460.9361} C_DIS
LIN {X 130.2276,Y -29.243,Z 181,A -10.1451,B 5.147,C 0.2575,E1 5.3093,E2 462.6079} C_DIS
LIN {X 129.295,Y -33.1214,Z 181,A -11.8256,B 5.1468,C 0.2618,E1 5.3081,E2 464.2858} C_DIS
LIN {X 128.1908,Y -37.1668,Z 181,A -13.702,B 5.1465,C 0.2678,E1 5.3067,E2 466.1731} C_DIS
LIN {X 126.9493,Y -41.2113,Z 181,A -15.3275,B 5.1464,C 0.2701,E1 5.3054,E2 467.7767} C_DIS
LIN {X 125.9052,Y -44.2985,Z 181,A -16.6911,B 5.1462,C 0.2734,E1 5.3041,E2 469.1371} C_DIS
LIN {X 124.8556,Y -47.1733,Z 181,A -17.991,B 5.146,C 0.2767,E1 5.3029,E2 470.4364} C_DIS
LIN {X 123.5816,Y -50.418,Z 181,A -19.431,B 5.1458,C 0.2799,E1 5.3014,E2 471.8708} C_DIS
LIN {X 122.3894,Y -53.2448,Z 181,A -20.7357,B 5.1457,C 0.2833,E1 5.2999,E2 473.175} C_DIS
LIN {X 120.9639,Y -56.4091,Z 181,A -22.286,B 5.1454,C 0.288,E1 5.2981,E2 474.7342} C_DIS
LIN {X 119.2249,Y -59.999,Z 181,A -23.8253,B 5.1453,C 0.29,E1 5.2962,E2 476.2535} C_DIS
LIN {X 117.7217,Y -62.8993,Z 181,A -25.3292,B 5.145,C 0.295,E1 5.2943,E2 477.7713} C_DIS
LIN {X 115.6699,Y -66.5973,Z 181,A -27.1035,B 5.1448,C 0.299,E1 5.2918,E2 479.5421} C_DIS
LIN {X 113.6302,Y -70.0205,Z 181,A -28.6455,B 5.1447,C 0.3009,E1 5.2896,E2 481.0646} C_DIS
LIN {X 111.8795,Y -72.7846,Z 181,A -30.0147,B 5.1445,C 0.3039,E1 5.2876,E2 482.4307} C_DIS
LIN {X 110.0603,Y -75.5072,Z 181,A -31.3886,B 5.1443,C 0.3068,E1 5.2854,E2 483.8019} C_DIS
LIN {X 108.1662,Y -78.1966,Z 181,A -32.7618,B 5.1441,C 0.3096,E1 5.2832,E2 485.1715} C_DIS
LIN {X 106.2178,Y -80.8239,Z 181,A -34.2144,B 5.1439,C 0.3136,E1 5.2807,E2 486.6314} C_DIS
LIN {X 103.6924,Y -84.0392,Z 181,A -35.9462,B 5.1437,C 0.3173,E1 5.2777,E2 488.3618} C_DIS
LIN {X 101.0542,Y -87.1933,Z 181,A -37.6357,B 5.1435,C 0.3202,E1 5.2747,E2 490.0434} C_DIS
LIN {X 98.3375,Y -90.2461,Z 181,A -39.3643,B 5.1433,C 0.3236,E1 5.2715,E2 491.7704} C_DIS
LIN {X 95.5281,Y -93.2153,Z 181,A -41.0944,B 5.1431,C 0.327,E1 5.2681,E2 493.499} C_DIS
LIN {X 92.629,Y -96.0967,Z 181,A -42.8315,B 5.1428,C 0.3304,E1 5.2647,E2 495.2353} C_DIS
LIN {X 89.6263,Y -98.9027,Z 181,A -44.5383,B 5.1427,C 0.3332,E1 5.2612,E2 496.9364} C_DIS
LIN {X 86.5552,Y -101.6013,Z 181,A -46.2715,B 5.1425,C 0.3363,E1 5.2575,E2 498.6684} C_DIS
LIN {X 83.403,Y -104.2049,Z 181,A -48.009,B 5.1423,C 0.3394,E1 5.2537,E2 500.4053} C_DIS
LIN {X 80.0753,Y -106.7835,Z 181,A -49.6938,B 5.1422,C 0.341,E1 5.25,E2 502.0763} C_DIS
LIN {X 77.6,Y -108.5949,Z 181,A -51.0165,B 5.142,C 0.3434,E1 5.247,E2 503.4007} C_DIS
LIN {X 74.7477,Y -110.5776,Z 181,A -52.448,B 5.1419,C 0.3452,E1 5.2437,E2 504.8259} C_DIS
LIN {X 72.0155,Y -112.3761,Z 181,A -53.8271,B 5.1417,C 0.3472,E1 5.2405,E2 506.2031} C_DIS
LIN {X 68.6255,Y -114.4782,Z 181,A -55.6507,B 5.1415,C 0.3513,E1 5.2361,E2 508.042} C_DIS
LIN {X 65.0016,Y -116.5743,Z 181,A -57.4338,B 5.1413,C 0.3538,E1 5.2318,E2 509.8248} C_DIS
LIN {X 61.4526,Y -118.4825,Z 181,A -58.9988,B 5.1413,C 0.3542,E1 5.228,E2 511.3703} C_DIS
LIN {X 58.5324,Y -119.9515,Z 181,A -60.3813,B 5.1412,C 0.3559,E1 5.2245,E2 512.7513} C_DIS
LIN {X 55.5767,Y -121.3488,Z 181,A -61.7651,B 5.141,C 0.3574,E1 5.221,E2 514.1337} C_DIS
LIN {X 52.5869,Y -122.6739,Z 181,A -63.1535,B 5.141,C 0.359,E1 5.2175,E2 515.5212} C_DIS
LIN {X 49.5446,Y -123.9337,Z 181,A -64.5463,B 5.1408,C 0.3604,E1 5.2139,E2 516.9123} C_DIS
LIN {X 46.5032,Y -125.1066,Z 181,A -65.9295,B 5.1408,C 0.3618,E1 5.2103,E2 518.2945} C_DIS
LIN {X 43.4337,Y -126.205,Z 181,A -67.3133,B 5.1407,C 0.3631,E1 5.2066,E2 519.6774} C_DIS
LIN {X 40.3093,Y -127.2375,Z 181,A -68.668,B 5.1407,C 0.3638,E1 5.203,E2 521.0258} C_DIS
LIN {X 37.1652,Y -128.1912,Z 181,A -70.2346,B 5.1404,C 0.367,E1 5.1988,E2 522.6128} C_DIS
LIN {X 33.12,Y -129.2953,Z 181,A -71.8976,B 5.1404,C 0.3668,E1 5.1943,E2 524.2598} C_DIS
LIN {X 29.9414,Y -130.0681,Z 181,A -73.4059,B 5.1402,C 0.3692,E1 5.1902,E2 525.782} C_DIS
LIN {X 26.0173,Y -130.9107,Z 181,A -74.9918,B 5.1402,C 0.3688,E1 5.1859,E2 527.3519} C_DIS
LIN {X 22.8018,Y -131.5095,Z 181,A -76.3852,B 5.1402,C 0.3695,E1 5.1821,E2 528.7448} C_DIS
LIN {X 19.7623,Y -132.0003,Z 181,A -77.7514,B 5.1402,C 0.3708,E1 5.1783,E2 530.1174} C_DIS
LIN {X 16.3363,Y -132.4673,Z 181,A -79.1971,B 5.1401,C 0.3711,E1 5.1743,E2 531.559} C_DIS
LIN {X 13.0501,Y -132.8306,Z 181,A -80.7225,B 5.1399,C 0.3729,E1 5.17,E2 533.0985} C_DIS
LIN {X 8.8691,Y -133.1765,Z 181,A -82.3412,B 5.1401,C 0.3714,E1 5.1656,E2 534.6953} C_DIS
LIN {X 4.9047,Y -133.3801,Z 181,A -84.2289,B 5.1399,C 0.3739,E1 5.1602,E2 536.6068} C_DIS
LIN {X 0.9666,Y -133.4651,Z 181,A -85.2273,B 5.1404,C 0.3663,E1 5.1577,E2 537.5188} C_DIS
Enddeposition()
LIN {X 0.9666,Y -133.4651,Z 181,A -85.2273,B 5.1404,C 0.3663,E1 5.1577,E2 537.5188} C_DIS
Startdeposition()
$VEL.CP = VEL_PRINT
LIN {X 3.2541,Y -134.3338,Z 181,A -84.0875,B 5.1405,C 0.3671,E1 5.1611,E2 536.3896} C_DIS
LIN {X 6.9391,Y -134.1931,Z 181,A -82.6145,B 5.1405,C 0.3679,E1 5.1651,E2 534.9286} C_DIS
LIN {X 12.1859,Y -133.8191,Z 181,A -80.1538,B 5.1407,C 0.3645,E1 5.172,E2 532.4388} C_DIS
LIN {X 17.3596,Y -133.2461,Z 181,A -78.134,B 5.1407,C 0.3659,E1 5.1776,E2 530.4433} C_DIS
LIN {X 20.8571,Y -132.7439,Z 181,A -76.5681,B 5.1407,C 0.3643,E1 5.1819,E2 528.869} C_DIS
LIN {X 26.2386,Y -131.7866,Z 181,A -74.3056,B 5.1407,C 0.3637,E1 5.1881,E2 526.6139} C_DIS
LIN {X 29.6997,Y -131.0489,Z 181,A -72.8514,B 5.1408,C 0.3632,E1 5.1921,E2 525.1657} C_DIS
LIN {X 33.0974,Y -130.2321,Z 181,A -71.3637,B 5.1408,C 0.3621,E1 5.1961,E2 523.6773} C_DIS
LIN {X 36.6702,Y -129.2724,Z 181,A -69.6958,B 5.1411,C 0.3596,E1 5.2006,E2 521.9969} C_DIS
LIN {X 40.6142,Y -128.0873,Z 181,A -68.0796,B 5.1411,C 0.3596,E1 5.2049,E2 520.3973} C_DIS
LIN {X 46.1605,Y -126.1958,Z 181,A -65.5717,B 5.1413,C 0.3569,E1 5.2115,E2 517.8866} C_DIS
LIN {X 52.5723,Y -123.6633,Z 181,A -62.6437,B 5.1415,C 0.3536,E1 5.2191,E2 514.9582} C_DIS
LIN {X 55.8935,Y -122.1965,Z 181,A -61.0111,B 5.1417,C 0.3505,E1 5.2233,E2 513.3136} C_DIS
LIN {X 59.6838,Y -120.3897,Z 181,A -59.3389,B 5.1417,C 0.3496,E1 5.2275,E2 511.6551} C_DIS
LIN {X 63.5227,Y -118.4111,Z 181,A -57.4785,B 5.1419,C 0.3468,E1 5.2321,E2 509.791} C_DIS
LIN {X 67.3371,Y -116.2842,Z 181,A -55.6451,B 5.1421,C 0.3443,E1 5.2365,E2 507.9598} C_DIS
LIN {X 71.0631,Y -114.0453,Z 181,A -53.8437,B 5.1423,C 0.3421,E1 5.2408,E2 506.1635} C_DIS
LIN {X 74.6283,Y -111.7449,Z 181,A -52.0596,B 5.1424,C 0.3394,E1 5.245,E2 504.3813} C_DIS
LIN {X 78.1172,Y -109.3344,Z 181,A -50.2804,B 5.1426,C 0.3367,E1 5.249,E2 502.6042} C_DIS
LIN {X 81.6263,Y -106.7401,Z 181,A -48.417,B 5.1428,C 0.3333,E1 5.2532,E2 500.7389} C_DIS
LIN {X 85.228,Y -103.8873,Z 181,A -46.4855,B 5.143,C 0.33,E1 5.2574,E2 498.8094} C_DIS
LIN {X 88.5393,Y -101.08,Z 181,A -44.6667,B 5.1432,C 0.3269,E1 5.2612,E2 496.9932} C_DIS
LIN {X 91.4394,Y -98.4641,Z 181,A -42.8766,B 5.1436,C 0.3218,E1 5.2649,E2 495.1856} C_DIS
LIN {X 95.2513,Y -94.7814,Z 181,A -40.8205,B 5.1436,C 0.3199,E1 5.269,E2 493.1536} C_DIS
LIN {X 98.3926,Y -91.5161,Z 181,A -38.9595,B 5.1439,C 0.3168,E1 5.2725,E2 491.3} C_DIS
LIN {X 100.6312,Y -89.0487,Z 181,A -37.4579,B 5.1441,C 0.3126,E1 5.2753,E2 489.7869} C_DIS
LIN {X 103.7525,Y -85.3926,Z 181,A -35.5046,B 5.1443,C 0.3093,E1 5.2788,E2 487.8441} C_DIS
LIN {X 106.4339,Y -82.026,Z 181,A -33.7581,B 5.1445,C 0.3063,E1 5.2818,E2 486.1072} C_DIS
LIN {X 109.0857,Y -78.465,Z 181,A -31.8602,B 5.1448,C 0.3018,E1 5.2849,E2 484.2071} C_DIS
LIN {X 111.661,Y -74.754,Z 181,A -30.0659,B 5.1449,C 0.299,E1 5.2877,E2 482.4278} C_DIS
LIN {X 113.7619,Y -71.5164,Z 181,A -28.3809,B 5.1452,C 0.2944,E1 5.2903,E2 480.7364} C_DIS
LIN {X 115.8812,Y -68.0283,Z 181,A -26.7323,B 5.1454,C 0.2914,E1 5.2926,E2 479.0978} C_DIS
LIN {X 118.0935,Y -64.1117,Z 181,A -24.7001,B 5.1457,C 0.2849,E1 5.2954,E2 477.0495} C_DIS
LIN {X 120.2679,Y -59.9306,Z 181,A -22.9035,B 5.1459,C 0.2828,E1 5.2976,E2 475.278} C_DIS
LIN {X 121.893,Y -56.5499,Z 181,A -21.5268,B 5.1459,C 0.2818,E1 5.2992,E2 473.9281} C_DIS
LIN {X 123.2419,Y -53.5468,Z 181,A -20.2348,B 5.146,C 0.2797,E1 5.3007,E2 472.6489} C_DIS
LIN {X 124.4595,Y -50.6539,Z 181,A -18.8582,B 5.1462,C 0.2756,E1 5.3022,E2 471.2664} C_DIS
LIN {X 125.8126,Y -47.1909,Z 181,A -17.2016,B 5.1465,C 0.2703,E1 5.3039,E2 469.5994} C_DIS
LIN {X 127.1765,Y -43.3864,Z 181,A -15.2722,B 5.1469,C 0.2627,E1 5.3057,E2 467.6425} C_DIS
LIN {X 128.6792,Y -38.7025,Z 181,A -13.4164,B 5.147,C 0.2604,E1 5.3072,E2 465.8154} C_DIS
LIN {X 129.7704,Y -34.8644,Z 181,A -11.7603,B 5.1472,C 0.2563,E1 5.3084,E2 464.1636} C_DIS
LIN {X 130.6645,Y -31.3469,Z 181,A -10.3289,B 5.1474,C 0.2537,E1 5.3093,E2 462.7455} C_DIS
LIN {X 131.5215,Y -27.5413,Z 181,A -8.6396,B 5.1476,C 0.2487,E1 5.3103,E2 461.0516} C_DIS
LIN {X 132.3794,Y -23.0637,Z 181,A -6.602,B 5.1479,C 0.2419,E1 5.3114,E2 459.0007} C_DIS
LIN {X 133.1347,Y -18.2099,Z 181,A -4.6913,B 5.1481,C 0.2386,E1 5.3121,E2 457.1114} C_DIS
LIN {X 133.5874,Y -14.5014,Z 181,A -3.1598,B 5.1483,C 0.235,E1 5.3126,E2 455.5863} C_DIS
LIN {X 133.9622,Y -10.5112,Z 181,A -1.5028,B 5.1484,C 0.2309,E1 5.313,E2 453.9345} C_DIS
LIN {X 134.1742,Y -7.3161,Z 181,A -0.0587,B 5.1487,C 0.2258,E1 5.3133,E2 452.4794} C_DIS
LIN {X 134.3474,Y -2.6139,Z 181,A 1.7899,B 5.1488,C 0.2224,E1 5.3133,E2 450.649} C_DIS
LIN {X 134.3658,Y 1.5035,Z 181,A 3.5745,B 5.149,C 0.217,E1 5.3133,E2 448.8596} C_DIS
LIN {X 134.2076,Y 6.6501,Z 181,A 5.6515,B 5.1492,C 0.2124,E1 5.3131,E2 446.7958} C_DIS
LIN {X 133.9279,Y 10.9253,Z 181,A 7.3913,B 5.1494,C 0.2085,E1 5.3128,E2 445.0655} C_DIS
LIN {X 133.5825,Y 14.5473,Z 181,A 8.881,B 5.1495,C 0.205,E1 5.3124,E2 443.5824} C_DIS
LIN {X 133.1357,Y 18.2022,Z 181,A 10.5106,B 5.1497,C 0.1997,E1 5.3118,E2 441.9444} C_DIS
LIN {X 132.5813,Y 21.8657,Z 181,A 11.9743,B 5.1498,C 0.1969,E1 5.3111,E2 440.494} C_DIS
LIN {X 131.9635,Y 25.3279,Z 181,A 13.4172,B 5.15,C 0.1935,E1 5.3104,E2 439.0571} C_DIS
LIN {X 131.1681,Y 29.1779,Z 181,A 15.1381,B 5.1502,C 0.1883,E1 5.3094,E2 437.3298} C_DIS
LIN {X 130.2942,Y 32.8525,Z 181,A 16.6035,B 5.1502,C 0.1859,E1 5.3084,E2 435.8813} C_DIS
LIN {X 129.4634,Y 35.9873,Z 181,A 17.975,B 5.1504,C 0.1822,E1 5.3074,E2 434.5104} C_DIS
LIN {X 128.4744,Y 39.3717,Z 181,A 19.4008,B 5.1504,C 0.1792,E1 5.3063,E2 433.0933} C_DIS
LIN {X 127.1424,Y 43.4846,Z 181,A 21.0863,B 5.1506,C 0.1765,E1 5.3048,E2 431.4263} C_DIS
LIN {X 126.185,Y 46.1906,Z 181,A 22.7964,B 5.1509,C 0.1664,E1 5.3031,E2 429.6553} C_DIS
LIN {X 124.8011,Y 49.8063,Z 181,A 24.3976,B 5.151,C 0.1627,E1 5.3015,E2 428.0594} C_DIS
LIN {X 123.3279,Y 53.3479,Z 181,A 25.6459,B 5.151,C 0.1639,E1 5.3001,E2 426.8582} C_DIS
LIN {X 121.4831,Y 57.4276,Z 181,A 27.5378,B 5.1511,C 0.1592,E1 5.2979,E2 424.9675} C_DIS
LIN {X 119.7206,Y 61.0143,Z 181,A 29.0936,B 5.1512,C 0.1569,E1 5.296,E2 423.4291} C_DIS
LIN {X 118.2706,Y 63.7842,Z 181,A 30.5088,B 5.1513,C 0.1524,E1 5.2941,E2 422.0033} C_DIS
LIN {X 116.1866,Y 67.5058,Z 181,A 32.2135,B 5.1514,C 0.1495,E1 5.2918,E2 420.3119} C_DIS
LIN {X 114.1366,Y 70.9165,Z 181,A 33.9167,B 5.1516,C 0.1453,E1 5.2893,E2 418.6072} C_DIS
LIN {X 111.9616,Y 74.3037,Z 181,A 35.5726,B 5.1516,C 0.142,E1 5.2868,E2 416.9582} C_DIS
LIN {X 109.7075,Y 77.5925,Z 181,A 37.248,B 5.1517,C 0.1384,E1 5.2841,E2 415.2851} C_DIS
LIN {X 107.064,Y 81.2016,Z 181,A 39.1583,B 5.1519,C 0.134,E1 5.2809,E2 413.3738} C_DIS
LIN {X 104.2762,Y 84.752,Z 181,A 41.0437,B 5.1519,C 0.1302,E1 5.2776,E2 411.4927} C_DIS
LIN {X 101.2848,Y 88.3046,Z 181,A 42.9724,B 5.152,C 0.1266,E1 5.2741,E2 409.5698} C_DIS
LIN {X 98.2328,Y 91.6878,Z 181,A 44.7169,B 5.152,C 0.1251,E1 5.2709,E2 407.849} C_DIS
LIN {X 95.4632,Y 94.568,Z 181,A 46.5561,B 5.1522,C 0.1198,E1 5.2673,E2 405.993} C_DIS
LIN {X 92.1129,Y 97.8342,Z 181,A 48.4575,B 5.1522,C 0.1171,E1 5.2635,E2 404.1026} C_DIS
LIN {X 88.0953,Y 101.4674,Z 181,A 50.7687,B 5.1524,C 0.1127,E1 5.2587,E2 401.7908} C_DIS
LIN {X 85.126,Y 103.9706,Z 181,A 52.3733,B 5.1524,C 0.1103,E1 5.2552,E2 400.1923} C_DIS
LIN {X 81.9465,Y 106.4952,Z 181,A 54.1189,B 5.1524,C 0.107,E1 5.2514,E2 398.4447} C_DIS
LIN {X 78.3356,Y 109.1782,Z 181,A 55.9918,B 5.1525,C 0.1044,E1 5.2471,E2 396.5773} C_DIS
LIN {X 74.6048,Y 111.7605,Z 181,A 57.8193,B 5.1525,C 0.1026,E1 5.243,E2 394.7626} C_DIS
LIN {X 71.1622,Y 113.9837,Z 181,A 59.6138,B 5.1526,C 0.0993,E1 5.2387,E2 392.9624} C_DIS
LIN {X 67.3663,Y 116.2673,Z 181,A 61.4247,B 5.1526,C 0.0975,E1 5.2344,E2 391.1609} C_DIS
LIN {X 63.6305,Y 118.3532,Z 181,A 63.2675,B 5.1527,C 0.0947,E1 5.2299,E2 389.316} C_DIS
LIN {X 59.7419,Y 120.361,Z 181,A 65.0254,B 5.1527,C 0.0935,E1 5.2255,E2 387.5712} C_DIS
LIN {X 56.4265,Y 121.9501,Z 181,A 66.5408,B 5.1527,C 0.0922,E1 5.2217,E2 386.0623} C_DIS
LIN {X 53.3026,Y 123.3475,Z 181,A 67.9569,B 5.1527,C 0.091,E1 5.2181,E2 384.6515} C_DIS
LIN {X 50.3116,Y 124.5975,Z 181,A 69.3527,B 5.1528,C 0.0893,E1 5.2145,E2 383.2542} C_DIS
LIN {X 47.244,Y 125.7927,Z 181,A 70.8117,B 5.1528,C 0.0872,E1 5.2107,E2 381.7888} C_DIS
LIN {X 43.1815,Y 127.2468,Z 181,A 72.5644,B 5.1528,C 0.0864,E1 5.2061,E2 380.047} C_DIS
LIN {X 40.0566,Y 128.264,Z 181,A 74.8467,B 5.1531,C 0.0747,E1 5.1997,E2 377.6581} C_DIS
LIN {X 33.9042,Y 130.0265,Z 181,A 76.732,B 5.1529,C 0.0825,E1 5.1949,E2 375.8759} C_DIS
LIN {X 30.1557,Y 130.9447,Z 181,A 78.251,B 5.1529,C 0.0828,E1 5.1908,E2 374.3725} C_DIS
LIN {X 27.2159,Y 131.5877,Z 181,A 79.5679,B 5.1529,C 0.0816,E1 5.1872,E2 373.052} C_DIS
LIN {X 23.8767,Y 132.2339,Z 181,A 80.9925,B 5.1529,C 0.0811,E1 5.1833,E2 371.6308} C_DIS
LIN {X 20.2592,Y 132.8364,Z 181,A 82.5922,B 5.1529,C 0.0799,E1 5.1789,E2 370.0273} C_DIS
LIN {X 16.2481,Y 133.3866,Z 181,A 84.3493,B 5.1529,C 0.0789,E1 5.174,E2 368.2671} C_DIS
LIN {X 13.3183,Y 133.7114,Z 181,A 85.7464,B 5.153,C 0.0769,E1 5.1701,E2 366.8537} C_DIS
LIN {X 8.533,Y 134.1013,Z 181,A 87.6509,B 5.153,C 0.078,E1 5.1648,E2 364.967} C_DIS
LIN {X 4.7719,Y 134.2883,Z 181,A 89.2168,B 5.153,C 0.0781,E1 5.1604,E2 363.4066} C_DIS
LIN {X 0.9592,Y 134.3691,Z 181,A 90.9006,B 5.153,C 0.0774,E1 5.1557,E2 361.7165} C_DIS
LIN {X -3.6846,Y 134.3218,Z 181,A 92.9018,B 5.153,C 0.0771,E1 5.1501,E2 359.7137} C_DIS
LIN {X -7.7824,Y 134.1476,Z 181,A 94.5999,B 5.153,C 0.0779,E1 5.1454,E2 358.0225} C_DIS
LIN {X -11.3426,Y 133.8926,Z 181,A 96.0488,B 5.153,C 0.0789,E1 5.1414,E2 356.5831} C_DIS
LIN {X -16.7776,Y 133.3224,Z 181,A 98.4953,B 5.153,C 0.0783,E1 5.1346,E2 354.124} C_DIS
LIN {X -20.5284,Y 132.7947,Z 181,A 100.0021,B 5.153,C 0.08,E1 5.1304,E2 352.631} C_DIS
LIN {X -24.0336,Y 132.2058,Z 181,A 101.6904,B 5.153,C 0.0789,E1 5.1257,E2 350.9228} C_DIS
LIN {X -28.0551,Y 131.411,Z 181,A 103.3008,B 5.153,C 0.0813,E1 5.1214,E2 349.33} C_DIS
LIN {X -31.6508,Y 130.5913,Z 181,A 104.8935,B 5.153,C 0.082,E1 5.117,E2 347.7358} C_DIS
LIN {X -35.2262,Y 129.6739,Z 181,A 106.6139,B 5.153,C 0.0816,E1 5.1124,E2 345.9988} C_DIS
LIN {X -38.2589,Y 128.8113,Z 181,A 108.2783,B 5.153,C 0.0795,E1 5.1078,E2 344.2967} C_DIS
LIN {X -42.0462,Y 127.6248,Z 181,A 109.3828,B 5.1529,C 0.0867,E1 5.1051,E2 343.264} C_DIS
LIN {X -50.2514,Y 124.6217,Z 181,A 113.3729,B 5.1529,C 0.0877,E1 5.0946,E2 339.245} C_DIS
LIN {X -54.6229,Y 122.7688,Z 181,A 115.3212,B 5.1529,C 0.0906,E1 5.0896,E2 337.3073} C_DIS
LIN {X -57.6651,Y 121.3696,Z 181,A 116.7343,B 5.1528,C 0.0924,E1 5.086,E2 335.8969} C_DIS
LIN {X -60.5967,Y 119.9331,Z 181,A 118.1674,B 5.1528,C 0.0938,E1 5.0824,E2 334.46} C_DIS
LIN {X -63.1769,Y 118.5963,Z 181,A 119.955,B 5.1528,C 0.0902,E1 5.0778,E2 332.6072} C_DIS
LIN {X -66.9077,Y 116.5324,Z 181,A 121.421,B 5.1528,C 0.096,E1 5.0744,E2 331.185} C_DIS
LIN {X -70.1331,Y 114.6197,Z 181,A 123.3956,B 5.1528,C 0.0949,E1 5.0696,E2 329.1664} C_DIS
LIN {X -73.6279,Y 112.407,Z 181,A 125.2557,B 5.1527,C 0.0967,E1 5.0652,E2 327.2959} C_DIS
LIN {X -77.3176,Y 109.9014,Z 181,A 126.748,B 5.1526,C 0.1034,E1 5.0619,E2 325.8546} C_DIS
LIN {X -80.9071,Y 107.2863,Z 181,A 128.6485,B 5.1525,C 0.1065,E1 5.0576,E2 323.9548} C_DIS
LIN {X -84.2792,Y 104.6581,Z 181,A 130.5119,B 5.1525,C 0.1094,E1 5.0535,E2 322.088} C_DIS
LIN {X -87.5938,Y 101.9002,Z 181,A 132.3862,B 5.1524,C 0.1124,E1 5.0495,E2 320.2109} C_DIS
LIN {X -90.8067,Y 99.0478,Z 181,A 134.2788,B 5.1524,C 0.1153,E1 5.0456,E2 318.3124} C_DIS
LIN {X -94.1336,Y 95.8914,Z 181,A 136.2443,B 5.1522,C 0.119,E1 5.0417,E2 316.3473} C_DIS
LIN {X -97.1589,Y 92.8248,Z 181,A 138.1087,B 5.1522,C 0.1225,E1 5.038,E2 314.4811} C_DIS
LIN {X -100.0515,Y 89.6995,Z 181,A 139.9701,B 5.1521,C 0.1259,E1 5.0345,E2 312.6157} C_DIS
LIN {X -102.8108,Y 86.5233,Z 181,A 141.8318,B 5.152,C 0.1292,E1 5.0311,E2 310.7475} C_DIS
LIN {X -105.6123,Y 83.0804,Z 181,A 143.7206,B 5.1519,C 0.1334,E1 5.0278,E2 308.8607} C_DIS
LIN {X -108.1524,Y 79.7459,Z 181,A 145.6,B 5.1518,C 0.1367,E1 5.0247,E2 306.9716} C_DIS
LIN {X -110.7105,Y 76.1545,Z 181,A 147.4883,B 5.1517,C 0.141,E1 5.0217,E2 305.084} C_DIS
LIN {X -114.2226,Y 70.7783,Z 181,A 150.3242,B 5.1515,C 0.1468,E1 5.0174,E2 302.2387} C_DIS
LIN {X -116.4063,Y 67.1263,Z 181,A 152.1337,B 5.1514,C 0.1512,E1 5.0148,E2 300.4314} C_DIS
LIN {X -118.483,Y 63.3888,Z 181,A 154.1195,B 5.1513,C 0.1545,E1 5.0121,E2 298.4274} C_DIS
LIN {X -120.9365,Y 58.5716,Z 181,A 156.3695,B 5.1511,C 0.1608,E1 5.0093,E2 296.186} C_DIS
LIN {X -122.3954,Y 55.4578,Z 181,A 157.9323,B 5.1511,C 0.1638,E1 5.0075,E2 294.6127} C_DIS
LIN {X -123.8629,Y 52.0949,Z 181,A 159.4438,B 5.1509,C 0.1683,E1 5.0059,E2 293.109} C_DIS
LIN {X -125.2096,Y 48.7682,Z 181,A 161.0424,B 5.1507,C 0.1718,E1 5.0042,E2 291.5034} C_DIS
LIN {X -127.0592,Y 43.7248,Z 181,A 163.3418,B 5.1505,C 0.1779,E1 5.002,E2 289.2048} C_DIS
LIN {X -128.261,Y 40.0689,Z 181,A 165.1264,B 5.1505,C 0.1812,E1 5.0005,E2 287.4042} C_DIS
LIN {X -129.2869,Y 36.6184,Z 181,A 166.6357,B 5.1503,C 0.1856,E1 4.9993,E2 285.8992} C_DIS
LIN {X -130.1722,Y 33.3331,Z 181,A 167.8877,B 5.1501,C 0.1912,E1 4.9985,E2 284.6727} C_DIS
LIN {X -130.9776,Y 30.0118,Z 181,A 169.6364,B 5.15,C 0.1929,E1 4.9973,E2 282.8896} C_DIS
LIN {X -131.7902,Y 26.2206,Z 181,A 171.4062,B 5.1499,C 0.1966,E1 4.9963,E2 281.1069} C_DIS
LIN {X -132.521,Y 22.2274,Z 181,A 173.1744,B 5.1497,C 0.2011,E1 4.9955,E2 279.3355} C_DIS
LIN {X -133.1754,Y 17.8989,Z 181,A 175.116,B 5.1495,C 0.2058,E1 4.9947,E2 277.3862} C_DIS
LIN {X -133.6831,Y 13.6125,Z 181,A 177.0229,B 5.1493,C 0.2105,E1 4.9941,E2 275.4727} C_DIS
LIN {X -134.0228,Y 9.6846,Z 181,A 178.657,B 5.1491,C 0.2156,E1 4.9938,E2 273.8455} C_DIS
LIN {X -134.2564,Y 5.5903,Z 181,A -179.4634,B 5.1489,C 0.2196,E1 4.9935,E2 271.9512} C_DIS
LIN {X -134.3675,Y 1.2954,Z 181,A -177.4977,B 5.1488,C 0.2237,E1 4.9935,E2 269.9704} C_DIS
LIN {X -134.3266,Y -3.5115,Z 181,A -175.6356,B 5.1484,C 0.231,E1 4.9935,E2 268.133} C_DIS
LIN {X -134.1986,Y -6.8297,Z 181,A -174.0354,B 5.1484,C 0.2336,E1 4.9937,E2 266.511} C_DIS
LIN {X -133.9302,Y -10.8981,Z 181,A -172.2755,B 5.1481,C 0.2383,E1 4.9941,E2 264.7498} C_DIS
LIN {X -133.5783,Y -14.5866,Z 181,A -170.6258,B 5.1479,C 0.2422,E1 4.9945,E2 263.0924} C_DIS
LIN {X -133.0716,Y -18.653,Z 181,A -168.816,B 5.1477,C 0.2466,E1 4.9952,E2 261.2761} C_DIS
LIN {X -132.4728,Y -22.516,Z 181,A -167.1849,B 5.1475,C 0.2516,E1 4.9959,E2 259.6506} C_DIS
LIN {X -131.7195,Y -26.5683,Z 181,A -165.3452,B 5.1473,C 0.2558,E1 4.9969,E2 257.8018} C_DIS
LIN {X -130.9777,Y -30.0115,Z 181,A -163.3968,B 5.1473,C 0.2563,E1 4.9982,E2 255.7987} C_DIS
LIN {X -130.0119,Y -33.9589,Z 181,A -161.9243,B 5.1469,C 0.2632,E1 4.9992,E2 254.3599} C_DIS
LIN {X -128.9862,Y -37.6613,Z 181,A -160.3887,B 5.1466,C 0.2685,E1 5.0003,E2 252.8379} C_DIS
LIN {X -127.9918,Y -40.9133,Z 181,A -158.8659,B 5.1464,C 0.2718,E1 5.0016,E2 251.3069} C_DIS
LIN {X -126.9009,Y -44.1813,Z 181,A -157.3888,B 5.1462,C 0.2757,E1 5.0029,E2 249.8296} C_DIS
LIN {X -125.7789,Y -47.2809,Z 181,A -155.8519,B 5.1461,C 0.2783,E1 5.0044,E2 248.2772} C_DIS
LIN {X -124.2179,Y -51.2447,Z 181,A -154.0054,B 5.1459,C 0.2828,E1 5.0064,E2 246.4279} C_DIS
LIN {X -122.909,Y -54.3095,Z 181,A -152.5228,B 5.1457,C 0.2859,E1 5.008,E2 244.9383} C_DIS
LIN {X -121.451,Y -57.4947,Z 181,A -151.2194,B 5.1454,C 0.2913,E1 5.0095,E2 243.6593} C_DIS
LIN {X -119.9125,Y -60.6374,Z 181,A -148.1069,B 5.1459,C 0.2812,E1 5.0138,E2 240.3427} C_DIS
LIN {X -115.5189,Y -68.6421,Z 181,A -145.4591,B 5.1448,C 0.3014,E1 5.0173,E2 237.8549} C_DIS
LIN {X -113.1834,Y -72.4281,Z 181,A -143.5334,B 5.1445,C 0.3056,E1 5.0201,E2 235.9264} C_DIS
LIN {X -110.4918,Y -76.472,Z 181,A -141.364,B 5.1443,C 0.3096,E1 5.0235,E2 233.7453} C_DIS
LIN {X -108.0137,Y -79.9343,Z 181,A -139.5012,B 5.1441,C 0.3132,E1 5.0266,E2 231.8773} C_DIS
LIN {X -105.3859,Y -83.3683,Z 181,A -137.6077,B 5.1439,C 0.3168,E1 5.0299,E2 229.978} C_DIS
LIN {X -102.5023,Y -86.8885,Z 181,A -135.6541,B 5.1436,C 0.3208,E1 5.0334,E2 228.0233} C_DIS
LIN {X -100.1073,Y -89.6372,Z 181,A -134.1098,B 5.1434,C 0.3241,E1 5.0362,E2 226.4807} C_DIS
LIN {X -97.155,Y -92.8289,Z 181,A -132.1955,B 5.1432,C 0.3272,E1 5.0399,E2 224.5592} C_DIS
LIN {X -94.0731,Y -95.9508,Z 181,A -130.3157,B 5.143,C 0.3308,E1 5.0436,E2 222.6786} C_DIS
LIN {X -90.9553,Y -98.9113,Z 181,A -128.4352,B 5.1428,C 0.3338,E1 5.0475,E2 220.7924} C_DIS
LIN {X -87.6721,Y -101.8327,Z 181,A -126.558,B 5.1426,C 0.3371,E1 5.0514,E2 218.9151} C_DIS
LIN {X -84.6438,Y -104.3641,Z 181,A -124.7922,B 5.1425,C 0.3392,E1 5.0552,E2 217.139} C_DIS
LIN {X -81.4838,Y -106.8491,Z 181,A -123.0563,B 5.1423,C 0.3418,E1 5.0591,E2 215.4005} C_DIS
LIN {X -77.994,Y -109.4225,Z 181,A -121.189,B 5.1421,C 0.3446,E1 5.0633,E2 213.531} C_DIS
LIN {X -74.6103,Y -111.7569,Z 181,A -119.4215,B 5.1419,C 0.347,E1 5.0674,E2 211.7617} C_DIS
LIN {X -70.9797,Y -114.0973,Z 181,A -117.5867,B 5.1417,C 0.3497,E1 5.0717,E2 209.9277} C_DIS
LIN {X -67.4716,Y -116.2063,Z 181,A -115.7627,B 5.1417,C 0.3513,E1 5.0761,E2 208.0938} C_DIS
LIN {X -63.7316,Y -118.2988,Z 181,A -113.8303,B 5.1416,C 0.3526,E1 5.0809,E2 206.1479} C_DIS
LIN {X -59.759,Y -120.3526,Z 181,A -112.031,B 5.1413,C 0.3559,E1 5.0854,E2 204.3621} C_DIS
LIN {X -56.3103,Y -122.0038,Z 181,A -110.4502,B 5.1412,C 0.3582,E1 5.0893,E2 202.7875} C_DIS
LIN {X -53.2626,Y -123.3648,Z 181,A -109.0261,B 5.1411,C 0.3596,E1 5.093,E2 201.3631} C_DIS
LIN {X -50.1682,Y -124.6553,Z 181,A -107.5142,B 5.1411,C 0.3602,E1 5.0969,E2 199.8405} C_DIS
LIN {X -46.1534,Y -126.1984,Z 181,A -105.7253,B 5.1409,C 0.3623,E1 5.1016,E2 198.0571} C_DIS
LIN {X -43.1668,Y -127.2517,Z 181,A -103.4388,B 5.1415,C 0.3534,E1 5.108,E2 195.6501} C_DIS
LIN {X -37.0807,Y -129.1562,Z 181,A -101.5873,B 5.1407,C 0.3646,E1 5.1126,E2 193.9096} C_DIS
LIN {X -33.3349,Y -130.1718,Z 181,A -99.9901,B 5.1407,C 0.3662,E1 5.1169,E2 192.3193} C_DIS
LIN {X -29.938,Y -130.9945,Z 181,A -98.4243,B 5.1407,C 0.3662,E1 5.1212,E2 190.7435} C_DIS
LIN {X -26.6939,Y -131.6939,Z 181,A -96.9353,B 5.1407,C 0.366,E1 5.1253,E2 189.2446} C_DIS
LIN {X -22.3971,Y -132.4927,Z 181,A -95.1739,B 5.1405,C 0.3678,E1 5.1301,E2 187.4956} C_DIS
LIN {X -19.1831,Y -132.9959,Z 181,A -93.7634,B 5.1405,C 0.368,E1 5.134,E2 186.0816} C_DIS
LIN {X -16.4086,Y -133.3675,Z 181,A -92.3637,B 5.1406,C 0.366,E1 5.138,E2 184.6552} C_DIS
LIN {X -11.2897,Y -133.8971,Z 181,A -90.3391,B 5.1405,C 0.3682,E1 5.1435,E2 182.6515} C_DIS
LIN {X -7.1836,Y -134.1808,Z 181,A -88.5562,B 5.1405,C 0.3679,E1 5.1485,E2 180.8642} C_DIS
LIN {X -4.0181,Y -134.3125,Z 181,A -87.1784,B 5.1405,C 0.3676,E1 5.1524,E2 179.4824} C_DIS
LIN {X 0.9637,Y -134.3675,Z 181,A -85.9688,B 5.1398,C 0.3779,E1 5.1555,E2 178.3881} C_DIS
Enddeposition()
LIN {X 0.9637,Y -134.3675,Z 181,A -85.9689,B 5.1398,C 0.3779,E1 5.1555,E2 178.3883} C_DIS
Startdeposition()
$VEL.CP = VEL_PRINT
LIN {X -3.8452,Y -135.22,Z 181,A -87.8416,B 5.1393,C 0.3791,E1 5.1498,E2 180.2738} C_DIS
LIN {X -8.1217,Y -135.0307,Z 181,A -89.6266,B 5.1393,C 0.3787,E1 5.1449,E2 182.0561} C_DIS
LIN {X -11.8391,Y -134.7563,Z 181,A -91.1308,B 5.1394,C 0.3777,E1 5.1407,E2 183.5513} C_DIS
LIN {X -18.6995,Y -133.9765,Z 181,A -94.1849,B 5.1394,C 0.3786,E1 5.1322,E2 186.6232} C_DIS
LIN {X -22.4759,Y -133.3944,Z 181,A -95.7074,B 5.1394,C 0.377,E1 5.128,E2 188.134} C_DIS
LIN {X -25.7834,Y -132.7951,Z 181,A -97.2801,B 5.1394,C 0.378,E1 5.1236,E2 189.7261} C_DIS
LIN {X -29.934,Y -131.921,Z 181,A -99.0081,B 5.1395,C 0.3764,E1 5.1189,E2 191.4459} C_DIS
LIN {X -33.5182,Y -131.0562,Z 181,A -100.5295,B 5.1396,C 0.3751,E1 5.1148,E2 192.9626} C_DIS
LIN {X -36.7282,Y -130.1932,Z 181,A -101.9572,B 5.1396,C 0.3744,E1 5.111,E2 194.3932} C_DIS
LIN {X -40.3922,Y -129.1051,Z 181,A -104.0342,B 5.1394,C 0.3781,E1 5.1053,E2 196.5286} C_DIS
LIN {X -44.1889,Y -127.8533,Z 181,A -105.2901,B 5.1398,C 0.3722,E1 5.1021,E2 197.7295} C_DIS
LIN {X -47.5471,Y -126.6428,Z 181,A -106.7385,B 5.14,C 0.3702,E1 5.0983,E2 199.1701} C_DIS
LIN {X -50.8319,Y -125.3606,Z 181,A -108.2858,B 5.14,C 0.3694,E1 5.0943,E2 200.7245} C_DIS
LIN {X -53.7865,Y -124.1214,Z 181,A -109.7117,B 5.14,C 0.3687,E1 5.0906,E2 202.1593} C_DIS
LIN {X -57.0374,Y -122.6617,Z 181,A -111.1883,B 5.1402,C 0.3668,E1 5.0869,E2 203.6319} C_DIS
LIN {X -60.0231,Y -121.2285,Z 181,A -112.6695,B 5.1402,C 0.366,E1 5.0831,E2 205.1232} C_DIS
LIN {X -63.5632,Y -119.4126,Z 181,A -114.3762,B 5.1404,C 0.3641,E1 5.0789,E2 206.8328} C_DIS
LIN {X -67.3655,Y -117.3102,Z 181,A -116.3264,B 5.1405,C 0.3629,E1 5.0741,E2 208.7969} C_DIS
LIN {X -71.2113,Y -115.016,Z 181,A -118.2193,B 5.1407,C 0.3602,E1 5.0696,E2 210.6894} C_DIS
LIN {X -74.9169,Y -112.6372,Z 181,A -120.1359,B 5.1408,C 0.358,E1 5.0651,E2 212.6125} C_DIS
LIN {X -78.5559,Y -110.13,Z 181,A -121.9963,B 5.141,C 0.355,E1 5.0608,E2 214.4713} C_DIS
LIN {X -82.004,Y -107.5873,Z 181,A -123.7995,B 5.1413,C 0.352,E1 5.0568,E2 216.273} C_DIS
LIN {X -85.2571,Y -105.0286,Z 181,A -125.666,B 5.1413,C 0.3501,E1 5.0527,E2 218.1536} C_DIS
LIN {X -88.9593,Y -101.9111,Z 181,A -127.7211,B 5.1416,C 0.3465,E1 5.0483,E2 220.2089} C_DIS
LIN {X -92.2471,Y -98.9449,Z 181,A -129.6823,B 5.1418,C 0.3438,E1 5.0443,E2 222.1806} C_DIS
LIN {X -95.634,Y -95.6762,Z 181,A -131.6879,B 5.1421,C 0.3401,E1 5.0403,E2 224.1873} C_DIS
LIN {X -98.7159,Y -92.493,Z 181,A -133.8133,B 5.1421,C 0.3386,E1 5.0361,E2 226.3435} C_DIS
LIN {X -101.0083,Y -89.9838,Z 181,A -135.058,B 5.1425,C 0.3339,E1 5.0339,E2 227.5635} C_DIS
LIN {X -103.9277,Y -86.5958,Z 181,A -137.0051,B 5.1427,C 0.3304,E1 5.0303,E2 229.5167} C_DIS
LIN {X -106.7222,Y -83.127,Z 181,A -138.9496,B 5.1429,C 0.3268,E1 5.0269,E2 231.4679} C_DIS
LIN {X -109.3699,Y -79.6112,Z 181,A -140.8154,B 5.1432,C 0.3227,E1 5.0238,E2 233.3333} C_DIS
LIN {X -111.8411,Y -76.1006,Z 181,A -142.5779,B 5.1435,C 0.3181,E1 5.0211,E2 235.0882} C_DIS
LIN {X -113.891,Y -72.9964,Z 181,A -144.3046,B 5.1436,C 0.3157,E1 5.0184,E2 236.8331} C_DIS
LIN {X -116.3713,Y -68.9743,Z 181,A -146.5145,B 5.1438,C 0.3127,E1 5.0152,E2 239.0682} C_DIS
LIN {X -119.9729,Y -62.4962,Z 181,A -149.4722,B 5.1443,C 0.3034,E1 5.0113,E2 242.0018} C_DIS
LIN {X -121.8816,Y -58.6867,Z 181,A -151.3795,B 5.1446,C 0.2998,E1 5.0089,E2 243.9211} C_DIS
LIN {X -123.5104,Y -55.1748,Z 181,A -152.9613,B 5.1448,C 0.2951,E1 5.0071,E2 245.4948} C_DIS
LIN {X -124.7683,Y -52.2684,Z 181,A -154.3768,B 5.145,C 0.2922,E1 5.0055,E2 246.9189} C_DIS
LIN {X -126.1779,Y -48.7678,Z 181,A -156.4086,B 5.145,C 0.2916,E1 5.0034,E2 249.0036} C_DIS
LIN {X -127.5219,Y -45.143,Z 181,A -157.6828,B 5.1454,C 0.2843,E1 5.0022,E2 250.2319} C_DIS
LIN {X -128.5401,Y -42.1538,Z 181,A -159.1151,B 5.1456,C 0.2815,E1 5.0009,E2 251.6753} C_DIS
LIN {X -129.753,Y -38.2536,Z 181,A -160.9421,B 5.1458,C 0.2776,E1 4.9994,E2 253.5131} C_DIS
LIN {X -131.0892,Y -33.3884,Z 181,A -163.2068,B 5.1461,C 0.2728,E1 4.9978,E2 255.7923} C_DIS
LIN {X -131.9569,Y -29.7767,Z 181,A -164.6677,B 5.1463,C 0.2676,E1 4.9969,E2 257.2384} C_DIS
LIN {X -132.5691,Y -26.9182,Z 181,A -165.9412,B 5.1465,C 0.2644,E1 4.9962,E2 258.5155} C_DIS
LIN {X -133.1859,Y -23.6796,Z 181,A -167.3614,B 5.1467,C 0.2607,E1 4.9955,E2 259.9377} C_DIS
LIN {X -133.7426,Y -20.3038,Z 181,A -168.9231,B 5.1468,C 0.2576,E1 4.9948,E2 261.5123} C_DIS
LIN {X -134.3182,Y -16.0569,Z 181,A -170.7638,B 5.1471,C 0.2527,E1 4.9941,E2 263.3549} C_DIS
LIN {X -134.7512,Y -11.8997,Z 181,A -172.6404,B 5.1473,C 0.2485,E1 4.9936,E2 265.2434} C_DIS
LIN {X -135.0398,Y -7.9742,Z 181,A -174.3008,B 5.1475,C 0.2437,E1 4.9933,E2 266.9018} C_DIS
LIN {X -135.2263,Y -3.62,Z 181,A -176.1681,B 5.1477,C 0.2386,E1 4.9931,E2 268.7703} C_DIS
LIN {X -135.2754,Y -0.2198,Z 181,A -177.7477,B 5.1479,C 0.2357,E1 4.9931,E2 270.3659} C_DIS
LIN {X -135.2218,Y 3.7818,Z 181,A -179.4011,B 5.1481,C 0.2305,E1 4.9931,E2 272.0129} C_DIS
LIN {X -135.0812,Y 7.245,Z 181,A 178.982,B 5.1482,C 0.2275,E1 4.9934,E2 273.647} C_DIS
LIN {X -134.7932,Y 11.4023,Z 181,A 177.3134,B 5.1485,C 0.2217,E1 4.9937,E2 275.3024} C_DIS
LIN {X -134.4791,Y 14.6498,Z 181,A 175.8522,B 5.1486,C 0.2184,E1 4.9941,E2 276.7722} C_DIS
LIN {X -134.0414,Y 18.2355,Z 181,A 174.1471,B 5.1488,C 0.2155,E1 4.9948,E2 278.4976} C_DIS
LIN {X -133.4443,Y 22.1765,Z 181,A 172.5036,B 5.149,C 0.2104,E1 4.9955,E2 280.1342} C_DIS
LIN {X -132.7219,Y 26.1664,Z 181,A 170.7975,B 5.1492,C 0.2055,E1 4.9964,E2 281.8375} C_DIS
LIN {X -132.1945,Y 28.702,Z 181,A 169.591,B 5.1492,C 0.2033,E1 4.9971,E2 283.0564} C_DIS
LIN {X -131.3505,Y 32.3517,Z 181,A 168.0333,B 5.1494,C 0.1987,E1 4.9981,E2 284.6094} C_DIS
LIN {X -130.4176,Y 35.9257,Z 181,A 166.5342,B 5.1496,C 0.1939,E1 4.9991,E2 286.0991} C_DIS
LIN {X -129.0524,Y 40.5586,Z 181,A 164.2025,B 5.1497,C 0.1906,E1 5.0011,E2 288.464} C_DIS
LIN {X -127.019,Y 46.538,Z 181,A 161.6047,B 5.15,C 0.1828,E1 5.0034,E2 291.0501} C_DIS
LIN {X -125.4692,Y 50.5626,Z 181,A 159.6318,B 5.1502,C 0.1791,E1 5.0054,E2 293.0392} C_DIS
LIN {X -124.0428,Y 53.9681,Z 181,A 158.0653,B 5.1502,C 0.175,E1 5.0072,E2 294.6047} C_DIS
LIN {X -122.5827,Y 57.2084,Z 181,A 156.4456,B 5.1504,C 0.172,E1 5.0091,E2 296.2369} C_DIS
LIN {X -119.3847,Y 63.6163,Z 181,A 153.597,B 5.1507,C 0.1629,E1 5.0126,E2 299.0607} C_DIS
LIN {X -118.049,Y 66.0615,Z 181,A 152.135,B 5.1507,C 0.1622,E1 5.0146,E2 300.5557} C_DIS
LIN {X -115.6534,Y 70.171,Z 181,A 149.8483,B 5.1507,C 0.1595,E1 5.018,E2 302.8734} C_DIS
LIN {X -113.9588,Y 72.8904,Z 181,A 148.6742,B 5.1509,C 0.1548,E1 5.0197,E2 304.0244} C_DIS
LIN {X -111.5364,Y 76.5457,Z 181,A 146.7639,B 5.1511,C 0.1508,E1 5.0227,E2 305.9394} C_DIS
LIN {X -109.0062,Y 80.1079,Z 181,A 144.8709,B 5.1511,C 0.1469,E1 5.0258,E2 307.836} C_DIS
LIN {X -106.225,Y 83.7612,Z 181,A 142.8751,B 5.1513,C 0.143,E1 5.0292,E2 309.8363} C_DIS
LIN {X -103.4527,Y 87.1621,Z 181,A 140.9716,B 5.1513,C 0.1393,E1 5.0326,E2 311.7435} C_DIS
LIN {X -100.4837,Y 90.5694,Z 181,A 138.9893,B 5.1515,C 0.1359,E1 5.0363,E2 313.7324} C_DIS
LIN {X -97.4228,Y 93.8538,Z 181,A 137.0394,B 5.1515,C 0.1324,E1 5.04,E2 315.6865} C_DIS
LIN {X -94.2483,Y 97.0409,Z 181,A 135.1038,B 5.1517,C 0.1288,E1 5.0439,E2 317.6242} C_DIS
LIN {X -90.8277,Y 100.2495,Z 181,A 133.1172,B 5.1517,C 0.1251,E1 5.0479,E2 319.6091} C_DIS
LIN {X -87.3679,Y 103.2791,Z 181,A 131.1153,B 5.1518,C 0.122,E1 5.0522,E2 321.6159} C_DIS
LIN {X -83.8802,Y 106.1315,Z 181,A 129.1396,B 5.1518,C 0.1192,E1 5.0565,E2 323.5982} C_DIS
LIN {X -80.3108,Y 108.8571,Z 181,A 127.2618,B 5.152,C 0.1158,E1 5.0607,E2 325.4715} C_DIS
LIN {X -76.7944,Y 111.3658,Z 181,A 125.4088,B 5.152,C 0.113,E1 5.0649,E2 327.3259} C_DIS
LIN {X -72.8405,Y 113.9907,Z 181,A 122.7654,B 5.152,C 0.1157,E1 5.0713,E2 330.043} C_DIS
LIN {X -68.3962,Y 116.7116,Z 181,A 121.1081,B 5.1521,C 0.1076,E1 5.0751,E2 331.6335} C_DIS
LIN {X -63.9475,Y 119.2072,Z 181,A 118.9221,B 5.1521,C 0.1049,E1 5.0805,E2 333.8208} C_DIS
LIN {X -61.0938,Y 120.6927,Z 181,A 117.633,B 5.1522,C 0.1025,E1 5.0837,E2 335.1001} C_DIS
LIN {X -58.1149,Y 122.1548,Z 181,A 116.2011,B 5.1522,C 0.101,E1 5.0873,E2 336.5341} C_DIS
LIN {X -54.7061,Y 123.7201,Z 181,A 114.282,B 5.1522,C 0.1024,E1 5.0923,E2 338.4916} C_DIS
LIN {X -51.6189,Y 125.0396,Z 181,A 113.182,B 5.1523,C 0.0978,E1 5.095,E2 339.5522} C_DIS
LIN {X -45.2215,Y 127.4927,Z 181,A 110.0379,B 5.1523,C 0.0974,E1 5.1033,E2 342.7233} C_DIS
LIN {X -41.7059,Y 128.6859,Z 181,A 108.4551,B 5.1523,C 0.0962,E1 5.1075,E2 344.3063} C_DIS
LIN {X -37.229,Y 130.053,Z 181,A 106.6257,B 5.1524,C 0.0931,E1 5.1123,E2 346.1163} C_DIS
LIN {X -33.4533,Y 131.0727,Z 181,A 104.9704,B 5.1524,C 0.092,E1 5.1168,E2 347.7703} C_DIS
LIN {X -30.1372,Y 131.8746,Z 181,A 103.4932,B 5.1524,C 0.0914,E1 5.1208,E2 349.2506} C_DIS
LIN {X -26.2011,Y 132.7151,Z 181,A 101.6874,B 5.1524,C 0.0916,E1 5.1258,E2 351.0675} C_DIS
LIN {X -22.2625,Y 133.43,Z 181,A 100.0878,B 5.1524,C 0.0898,E1 5.1302,E2 352.6547} C_DIS
LIN {X -18.6932,Y 133.9774,Z 181,A 98.5278,B 5.1524,C 0.0896,E1 5.1345,E2 354.2175} C_DIS
LIN {X -13.0449,Y 134.6442,Z 181,A 96.0654,B 5.1524,C 0.0896,E1 5.1413,E2 356.685} C_DIS
LIN {X -8.1973,Y 135.0261,Z 181,A 94.1011,B 5.1525,C 0.0882,E1 5.1468,E2 358.6369} C_DIS
LIN {X -4.091,Y 135.2132,Z 181,A 91.9014,B 5.1525,C 0.093,E1 5.1531,E2 360.8904} C_DIS
LIN {X 0.0644,Y 135.276,Z 181,A 90.275,B 5.1525,C 0.0916,E1 5.1576,E2 362.5002} C_DIS
LIN {X 3.3832,Y 135.2329,Z 181,A 89.3384,B 5.1525,C 0.0867,E1 5.16,E2 363.3802} C_DIS
LIN {X 6.6116,Y 135.1131,Z 181,A 87.7892,B 5.1525,C 0.0889,E1 5.1644,E2 364.9505} C_DIS
LIN {X 10.5517,Y 134.8643,Z 181,A 85.6063,B 5.1524,C 0.0949,E1 5.1707,E2 367.1935} C_DIS
LIN {X 15.128,Y 134.4276,Z 181,A 84.2641,B 5.1524,C 0.0889,E1 5.1742,E2 368.4631} C_DIS
LIN {X 19.2228,Y 133.9017,Z 181,A 82.4733,B 5.1524,C 0.0901,E1 5.1792,E2 370.2583} C_DIS
LIN {X 23.0597,Y 133.2968,Z 181,A 80.7177,B 5.1524,C 0.0922,E1 5.184,E2 372.0267} C_DIS
LIN {X 26.8127,Y 132.5906,Z 181,A 79.1709,B 5.1524,C 0.0923,E1 5.1882,E2 373.5645} C_DIS
LIN {X 30.2797,Y 131.842,Z 181,A 77.7249,B 5.1524,C 0.0927,E1 5.1922,E2 375.0033} C_DIS
LIN {X 33.5796,Y 131.0407,Z 181,A 76.3001,B 5.1524,C 0.0936,E1 5.196,E2 376.4262} C_DIS
LIN {X 37.2514,Y 130.0465,Z 181,A 74.2387,B 5.1523,C 0.1002,E1 5.2017,E2 378.541} C_DIS
LIN {X 41.1339,Y 128.8686,Z 181,A 72.9574,B 5.1523,C 0.0966,E1 5.205,E2 379.7697} C_DIS
LIN {X 44.5424,Y 127.7308,Z 181,A 71.4659,B 5.1523,C 0.0976,E1 5.2089,E2 381.2573} C_DIS
Enddeposition()
END
